(**************************************DIAGNOSTICS**************************************)
(**************************************DIAGNOSTICS**************************************)
(**************************************DIAGNOSTICS**************************************)
	220:// Set Parameters to read the Diagnostic data of the AX5805.		
		IF i_nChooseChannel=1 THEN
			fbCoERead.nSubIndex:=16#07;
		ELSIF
			i_nChooseChannel=2 THEN
			fbCoERead.nSubIndex:=16#08;
		END_IF
		
			fbCoERead.nIndex	:= 	16#FA10;
			fbCoERead.pDstBuf	:= 	ADR(q_stAX5805_Diag.iDiagIndex);
			fbCoERead.cbBufLen	:= 	SIZEOF(q_stAX5805_Diag.iDiagIndex);
			fbCoERead.bExecute	:= 	TRUE;
			iState := iState + 10;	
			
	230:// Evaluate the Diagnostic data of the AX5805.		
		IF NOT fbCoERead.bBusy THEN
			IF q_stAX5805_Diag.iDiagIndex= 0 THEN
				q_stAX5805_Diag.sDiagReaction:='No Error Reaction.';
				ELSIF (q_stAX5805_Diag.iDiagIndex.4 AND q_stAX5805_Diag.iDiagIndex.6) THEN
					q_stAX5805_Diag.sDiagReaction:='SS1 (Safe Stop 1).';
				ELSIF q_stAX5805_Diag.iDiagIndex.6 THEN
					q_stAX5805_Diag.sDiagReaction:='STO (Safe Torque Off).';
				ELSE
					q_stAX5805_Diag.sDiagReaction:='Unknown.';
			END_IF
			
			IF q_stAX5805_Diag.iDiagIndex<255 THEN
				q_stAX5805_Diag.sDiagReason:='No error.';
				ELSIF (q_stAX5805_Diag.iDiagIndex.8 AND q_stAX5805_Diag.iDiagIndex.12 AND q_stAX5805_Diag.iDiagIndex.14 AND q_stAX5805_Diag.iDiagIndex.15) THEN
					q_stAX5805_Diag.sDiagReason:='The Safety Function SDIn has been turned off.';
				ELSIF (q_stAX5805_Diag.iDiagIndex.12 AND q_stAX5805_Diag.iDiagIndex.14 AND q_stAX5805_Diag.iDiagIndex.15) THEN
					q_stAX5805_Diag.sDiagReason:='The Safety Function SDIp has been turned off.';
				ELSIF (q_stAX5805_Diag.iDiagIndex.11 AND q_stAX5805_Diag.iDiagIndex.14 AND q_stAX5805_Diag.iDiagIndex.15) THEN
					q_stAX5805_Diag.sDiagReason:='The Safety Function SMA has been turned off.';
				ELSIF (q_stAX5805_Diag.iDiagIndex.14 AND q_stAX5805_Diag.iDiagIndex.15) THEN
					q_stAX5805_Diag.sDiagReason:='The Safety Function SAR has been turned off.';
				ELSIF (q_stAX5805_Diag.iDiagIndex.11 AND q_stAX5805_Diag.iDiagIndex.12 AND q_stAX5805_Diag.iDiagIndex.13 AND q_stAX5805_Diag.iDiagIndex.15) THEN
					q_stAX5805_Diag.sDiagReason:='The Safety Function SLI has been turned off.';
				ELSIF (q_stAX5805_Diag.iDiagIndex.11 AND q_stAX5805_Diag.iDiagIndex.13 AND q_stAX5805_Diag.iDiagIndex.15) THEN
					q_stAX5805_Diag.sDiagReason:='The Safety Function SMS has been turned off.';
				ELSIF (q_stAX5805_Diag.iDiagIndex.13 AND q_stAX5805_Diag.iDiagIndex.15) THEN
					q_stAX5805_Diag.sDiagReason:='The Safety Function SLP has been turned off.';
				ELSIF (q_stAX5805_Diag.iDiagIndex.12 AND q_stAX5805_Diag.iDiagIndex.15) THEN
					q_stAX5805_Diag.sDiagReason:='The Safety Function SLS has been turned off.';
				ELSIF (q_stAX5805_Diag.iDiagIndex.15) THEN
					q_stAX5805_Diag.sDiagReason:='The Safety Function SSR has been turned off.';
				ELSIF (q_stAX5805_Diag.iDiagIndex.11 AND q_stAX5805_Diag.iDiagIndex.13 AND q_stAX5805_Diag.iDiagIndex.14) THEN
					q_stAX5805_Diag.sDiagReason:='The Safety Function SOS has been turned off.';
				ELSIF (q_stAX5805_Diag.iDiagIndex.12 AND q_stAX5805_Diag.iDiagIndex.14) THEN
					q_stAX5805_Diag.sDiagReason:='The Safety Function SS1 has been turned off.';
				ELSIF (q_stAX5805_Diag.iDiagIndex.11) THEN
					q_stAX5805_Diag.sDiagReason:='The maximum traversing range was exceeded.';
				ELSIF (q_stAX5805_Diag.iDiagIndex.8 AND q_stAX5805_Diag.iDiagIndex.9 AND q_stAX5805_Diag.iDiagIndex.10) THEN
					q_stAX5805_Diag.sDiagReason:='Reason for shutdown position detection: External Cam detected to the left of the cam window.';
				ELSIF (q_stAX5805_Diag.iDiagIndex.9 AND q_stAX5805_Diag.iDiagIndex.10) THEN
					q_stAX5805_Diag.sDiagReason:='Reason for shutdown position detection: External Cam detected to the right of the cam window.';
				ELSIF (q_stAX5805_Diag.iDiagIndex.8 AND q_stAX5805_Diag.iDiagIndex.10) THEN
					q_stAX5805_Diag.sDiagReason:='Reason for shutdown position detection: External Cam detected unexpectedly.';
				ELSIF (q_stAX5805_Diag.iDiagIndex.10) THEN
					q_stAX5805_Diag.sDiagReason:='Internal comparison has failed. Please check the motor and drive dimensioning and parameterization.';
				ELSIF (q_stAX5805_Diag.iDiagIndex.8 AND q_stAX5805_Diag.iDiagIndex.9) THEN
					q_stAX5805_Diag.sDiagReason:='The FSOE Protocol is not in the DATA state.';
				ELSIF (q_stAX5805_Diag.iDiagIndex.9) THEN
					q_stAX5805_Diag.sDiagReason:='The parameters are incorrect or have not been loaded.';
				ELSIF (q_stAX5805_Diag.iDiagIndex.8) THEN
					q_stAX5805_Diag.sDiagReason:='The Status word was calculated incorrectly.';
				ELSIF (i_nChooseChannel<>1 AND i_nChooseChannel<>2) THEN
					q_stAX5805_Diag.sDiagReason:='Wrong Channel Number.';
				ELSE
					q_stAX5805_Diag.sDiagReason:= 'Unknown.';
			END_IF
			
			IF q_stAX5805_Diag.iDiagIndex = 0 THEN
				q_stAX5805_Diag.xDiagnosticAlarm := FALSE;
				ELSE
					q_stAX5805_Diag.xDiagnosticAlarm := TRUE;
			END_IF	
			fbCoERead.bExecute := FALSE;
			q_sErrorDescription := 'No Error';
			iState := iState + 10;
			IF fbCoERead.bError THEN
				q_sErrorDescription := 'AX5805 Diagnostic Data - Read Error';
			END_IF
		END_IF


(**************************************ERRORS**************************************)
(**************************************ERRORS**************************************)
(**************************************ERRORS**************************************)
	240:// Set Parameters to read the Error data of the AX5805.		
		IF i_nChooseChannel=1 THEN
			fbCoERead.nSubIndex:=16#03;
		ELSIF
			i_nChooseChannel=2 THEN
			fbCoERead.nSubIndex:=16#04;
		END_IF
		
			fbCoERead.nIndex	:= 	16#FA82;
			fbCoERead.pDstBuf	:= 	ADR(q_stAX5805_Diag.iErrorIndex);
			fbCoERead.cbBufLen	:= 	SIZEOF(q_stAX5805_Diag.iErrorIndex);
			fbCoERead.bExecute	:= 	TRUE;
			iState := iState + 10;	
			
	250:// Evaluate the Error data of the AX5805.	
		IF NOT fbCoERead.bBusy THEN	
			//0x0000
			IF q_stAX5805_Diag.iErrorIndex = 0 THEN
				q_stAX5805_Diag.sErrorName := 'No Error';
				q_stAX5805_Diag.sErrorDescription := 'No Error';
			//0x0001
			ELSIF q_stAX5805_Diag.iErrorIndex = 16#0001 THEN
				q_stAX5805_Diag.sErrorName := 'FAULT_MAXT_C1';
				q_stAX5805_Diag.sErrorDescription := 'The temperature has exceeded the maximum permissible temperature (MC1).';
				q_stAX5805_Diag.xMC1_TempHighAlarm := TRUE;
			//0x0002
			ELSIF q_stAX5805_Diag.iErrorIndex = 16#0002 THEN
				q_stAX5805_Diag.sErrorName := 'FAULT_MAXT_C2';
				q_stAX5805_Diag.sErrorDescription := 'The temperature has exceeded the maximum permissible temperature (MC2).';
				q_stAX5805_Diag.xMC2_TempHighAlarm := TRUE;
			//0x0003
			ELSIF q_stAX5805_Diag.iErrorIndex = 16#0003 THEN
				q_stAX5805_Diag.sErrorName := 'FAULT_MINT_C1';
				q_stAX5805_Diag.sErrorDescription := 'The temperature has fallen below the minimum permissible temperature (MC1).';
				q_stAX5805_Diag.xMC1_TempLowAlarm := TRUE;
			//0x0004
			ELSIF q_stAX5805_Diag.iErrorIndex = 16#0004 THEN
				q_stAX5805_Diag.sErrorName := 'FAULT_MINT_C2';
				q_stAX5805_Diag.sErrorDescription := 'The temperature has fallen below the minimum permissible temperature (MC2).';
				q_stAX5805_Diag.xMC2_TempLowAlarm := TRUE;	
			//0x0101
			ELSIF q_stAX5805_Diag.iErrorIndex = 16#0101 THEN
				q_stAX5805_Diag.sErrorName := 'HW_ERR_MAX_VCC_C1';
				q_stAX5805_Diag.sErrorDescription := 'The supply voltage has exceeded the maximum permissible voltage MC1 (3.3v).';
				q_stAX5805_Diag.xMC1_SupplyVoltHighAlarm := TRUE;
			//0x0102
			ELSIF q_stAX5805_Diag.iErrorIndex = 16#0102 THEN
				q_stAX5805_Diag.sErrorName := 'HW_ERR_MAX_VCC_C2';
				q_stAX5805_Diag.sErrorDescription := 'The supply voltage has exceeded the maximum permissible voltage MC2 (3.3v).';
				q_stAX5805_Diag.xMC2_SupplyVoltHighAlarm := TRUE;
			//0x0103
			ELSIF q_stAX5805_Diag.iErrorIndex = 16#0103 THEN
				q_stAX5805_Diag.sErrorName := 'HW_ERR_MIN_VCC_C1';
				q_stAX5805_Diag.sErrorDescription := 'The supply voltage has fallen below the minimum permissible voltage MC1 (3.3v).';
				q_stAX5805_Diag.xMC1_SupplyVoltLowAlarm := TRUE;
			//0x0104
			ELSIF q_stAX5805_Diag.iErrorIndex = 16#0104 THEN
				q_stAX5805_Diag.sErrorName := 'HW_ERR_MIN_VCC_C2';
				q_stAX5805_Diag.sErrorDescription := 'The supply voltage has fallen below the minimum permissible voltage MC2 (3.3v).';
				q_stAX5805_Diag.xMC2_SupplyVoltLowAlarm := TRUE;
				
			//0x0201
			ELSIF q_stAX5805_Diag.iErrorIndex = 16#0201 THEN
				q_stAX5805_Diag.sErrorName := 'FAULT_MCTC1_TO';
				q_stAX5805_Diag.sErrorDescription := 'The MCTests of MC1 were not carried out completely within the specified time.';
			//0x0202
			ELSIF q_stAX5805_Diag.iErrorIndex = 16#0202 THEN
				q_stAX5805_Diag.sErrorName := 'FAULT_MCTC2_TO';
				q_stAX5805_Diag.sErrorDescription := 'The MCTests of MC2 were not carried out completely within the specified time.';
			//0x0203
			ELSIF q_stAX5805_Diag.iErrorIndex = 16#0203 THEN
				q_stAX5805_Diag.sErrorName := 'FAULT_TIMER_C1';
				q_stAX5805_Diag.sErrorDescription := 'The global timer was not updated in time MC1.';
			//0x0204
			ELSIF q_stAX5805_Diag.iErrorIndex = 16#0204 THEN
				q_stAX5805_Diag.sErrorName := 'FAULT_TIMER_C2';
				q_stAX5805_Diag.sErrorDescription := 'The global timer was not updated in time MC2.';
			//0x20C
			ELSIF q_stAX5805_Diag.iErrorIndex = 16#020C THEN
				q_stAX5805_Diag.sErrorName := 'FAULT_TS_WDG_TO_C1';
				q_stAX5805_Diag.sErrorDescription := 'The TS module was not called within the watchdog time MC1.';
			//0x020D
			ELSIF q_stAX5805_Diag.iErrorIndex = 16#020D THEN
				q_stAX5805_Diag.sErrorName := 'FAULT_TS_WDG_TO_C2';
				q_stAX5805_Diag.sErrorDescription := 'The TwinSAFE module was not called within the watchdog time MC2.';
			//0x020E
			ELSIF q_stAX5805_Diag.iErrorIndex = 16#020E THEN
				q_stAX5805_Diag.sErrorName := 'FAULT_RESET_MC1';
				q_stAX5805_Diag.sErrorDescription := 'A reset has occurred in the operation of the controller for MC1. MC2 was not reset thereby.';
				
			//0x0300
			ELSIF q_stAX5805_Diag.iErrorIndex = 16#0300 THEN
				q_stAX5805_Diag.sErrorName := 'FAULT_SERCOMC2';
				q_stAX5805_Diag.sErrorDescription := 'Error group: an error occurred in the SerComP24C2 module during data transmission.';
				
			//0x0401
			ELSIF q_stAX5805_Diag.iErrorIndex = 16#0401 THEN
				q_stAX5805_Diag.sErrorName := 'FAULT_SERCOM';
				q_stAX5805_Diag.sErrorDescription := 'Error group: an error occurred in the SerComP24C1 module during data transmission.';
			//0x0402
			ELSIF q_stAX5805_Diag.iErrorIndex = 16#0402 THEN
				q_stAX5805_Diag.sErrorName := 'FAULT_SERCOM';
				q_stAX5805_Diag.sErrorDescription := 'Error group: an error occurred in the SerComP24C1 module during data transmission.';
			//0x0403
			ELSIF q_stAX5805_Diag.iErrorIndex = 16#0403 THEN
				q_stAX5805_Diag.sErrorName := 'FAULT_SERCOM';
				q_stAX5805_Diag.sErrorDescription := 'Error group: an error occurred in the SerComP24C1 module during data transmission.';
			//0x0404
			ELSIF q_stAX5805_Diag.iErrorIndex = 16#0404 THEN
				q_stAX5805_Diag.sErrorName := 'FAULT_SERCOM';
				q_stAX5805_Diag.sErrorDescription := 'Error group: an error occurred in the SerComP24C1 module during data transmission.';
			//0x0405
			ELSIF q_stAX5805_Diag.iErrorIndex = 16#0405 THEN
				q_stAX5805_Diag.sErrorName := 'FAULT_SERCOM';
				q_stAX5805_Diag.sErrorDescription := 'Error group: an error occurred in the SerComP24C1 module during data transmission.';
			//0x0406
			ELSIF q_stAX5805_Diag.iErrorIndex = 16#0406 THEN
				q_stAX5805_Diag.sErrorName := 'FAULT_SERCOM';
				q_stAX5805_Diag.sErrorDescription := 'Error group: an error occurred in the SerComP24C1 module during data transmission.';
			//0x0407
			ELSIF q_stAX5805_Diag.iErrorIndex = 16#0407 THEN
				q_stAX5805_Diag.sErrorName := 'FAULT_SERCOM';
				q_stAX5805_Diag.sErrorDescription := 'Error group: an error occurred in the SerComP24C1 module during data transmission.';
			//0x0408
			ELSIF q_stAX5805_Diag.iErrorIndex = 16#0408 THEN
				q_stAX5805_Diag.sErrorName := 'FAULT_SERCOM';
				q_stAX5805_Diag.sErrorDescription := 'Error group: an error occurred in the SerComP24C1 module during data transmission.';
			//0x0409
			ELSIF q_stAX5805_Diag.iErrorIndex = 16#0409 THEN
				q_stAX5805_Diag.sErrorName := 'FAULT_SERCOM';
				q_stAX5805_Diag.sErrorDescription := 'Error group: an error occurred in the SerComP24C1 module during data transmission.';
			//0x040A
			ELSIF q_stAX5805_Diag.iErrorIndex = 16#040A THEN
				q_stAX5805_Diag.sErrorName := 'FAULT_SERCOM';
				q_stAX5805_Diag.sErrorDescription := 'Error group: an error occurred in the SerComP24C1 module during data transmission.';
			//0x040B
			ELSIF q_stAX5805_Diag.iErrorIndex = 16#040B THEN
				q_stAX5805_Diag.sErrorName := 'FAULT_SERCOM';
				q_stAX5805_Diag.sErrorDescription := 'Error group: an error occurred in the SerComP24C1 module during data transmission.';
			//0x0501
			ELSIF q_stAX5805_Diag.iErrorIndex = 16#0501 THEN
				q_stAX5805_Diag.sErrorName := 'FAULT_TEMPSENSOR';
				q_stAX5805_Diag.sErrorDescription := 'Error in the communication with one of the temperature sensors.';
			//0x0502
			ELSIF q_stAX5805_Diag.iErrorIndex = 16#0502 THEN
				q_stAX5805_Diag.sErrorName := 'FAULT_TEMPSENSOR';
				q_stAX5805_Diag.sErrorDescription := 'Error in the communication with one of the temperature sensors.';
			//0x0503
			ELSIF q_stAX5805_Diag.iErrorIndex = 16#0503 THEN
				q_stAX5805_Diag.sErrorName := 'FAULT_TEMPSENSOR';
				q_stAX5805_Diag.sErrorDescription := 'Error in the communication with one of the temperature sensors..';
			//0x0504
			ELSIF q_stAX5805_Diag.iErrorIndex = 16#0504 THEN
				q_stAX5805_Diag.sErrorName := 'FAULT_TEMPSENSOR';
				q_stAX5805_Diag.sErrorDescription := 'Error in the communication with one of the temperature sensors.';
			//0x0505
			ELSIF q_stAX5805_Diag.iErrorIndex = 16#0505 THEN
				q_stAX5805_Diag.sErrorName := 'FAULT_TEMPSENSOR';
				q_stAX5805_Diag.sErrorDescription := 'Error in the communication with one of the temperature sensors.';
			//0x0506
			ELSIF q_stAX5805_Diag.iErrorIndex = 16#0506 THEN
				q_stAX5805_Diag.sErrorName := 'FAULT_TEMPSENSOR';
				q_stAX5805_Diag.sErrorDescription := 'Error in the communication with one of the temperature sensors.';
			//0x0507
			ELSIF q_stAX5805_Diag.iErrorIndex = 16#0507 THEN
				q_stAX5805_Diag.sErrorName := 'FAULT_TEMPSENSOR';
				q_stAX5805_Diag.sErrorDescription := 'Error in the communication with one of the temperature sensors.';
			//0x0601
			ELSIF q_stAX5805_Diag.iErrorIndex = 16#0601 THEN
				q_stAX5805_Diag.sErrorName := 'FAULT_OUTPUTCOMPARE';
				q_stAX5805_Diag.sErrorDescription := 'The values output by MC1 and MC2 differ.';
			//0x0602
			ELSIF q_stAX5805_Diag.iErrorIndex = 16#0602 THEN
				q_stAX5805_Diag.sErrorName := 'FAULT_OUTPUTCOMPAREC2';
				q_stAX5805_Diag.sErrorDescription := 'The values output by MC1 and MC2 differ.';
			//0x0700
			ELSIF q_stAX5805_Diag.iErrorIndex = 16#0700 THEN
				q_stAX5805_Diag.sErrorName := 'HW_ERR_MIN_VCC_FPGA';
				q_stAX5805_Diag.sErrorDescription := 'The FPGA supply voltage has fallen below the minimum value (5v).';
			//0x0701
			ELSIF q_stAX5805_Diag.iErrorIndex = 16#0701 THEN
				q_stAX5805_Diag.sErrorName := 'HW_ERR_MAX_VCC_FPGA';
				q_stAX5805_Diag.sErrorDescription := 'The FPGA supply voltage has exceeded the maximum value (5v).';
			//0x0710
			ELSIF q_stAX5805_Diag.iErrorIndex = 16#0710 THEN
				q_stAX5805_Diag.sErrorName := 'FAULT_FEEDBACK_C1';
				q_stAX5805_Diag.sErrorDescription := 'An error was detected in the feedback channels of MC1.';
			//0x0711
			ELSIF q_stAX5805_Diag.iErrorIndex = 16#0711 THEN
				q_stAX5805_Diag.sErrorName := 'FAULT_FEEDBACK_C2';
				q_stAX5805_Diag.sErrorDescription := 'An error was detected in the feedback channels of MC2.';
			//0x0720
			ELSIF q_stAX5805_Diag.iErrorIndex = 16#0720 THEN
				q_stAX5805_Diag.sErrorName := 'FAULT_Parameter_C1';
				q_stAX5805_Diag.sErrorDescription := 'General parameter error MC1.';
			//0x0721
			ELSIF q_stAX5805_Diag.iErrorIndex = 16#0721 THEN
				q_stAX5805_Diag.sErrorName := 'FAULT_Parameter_C2';
				q_stAX5805_Diag.sErrorDescription := 'General parameter error MC2.';
			//0x0722
			ELSIF q_stAX5805_Diag.iErrorIndex = 16#0722 THEN
				q_stAX5805_Diag.sErrorName := 'FAULT_Parameter_C1_DRIVE_PROFILE';
				q_stAX5805_Diag.sErrorDescription := 'Parameter: unkown parameter index MC1 drive profile.';
			//0x0723
			ELSIF q_stAX5805_Diag.iErrorIndex = 16#0723 THEN
				q_stAX5805_Diag.sErrorName := 'FAULT_Parameter_C1_VENDOR_SPECIFIC';
				q_stAX5805_Diag.sErrorDescription := 'Parameter: unkown parameter index MC1 vendor-specific.';
			//0x0724
			ELSIF q_stAX5805_Diag.iErrorIndex = 16#0724 THEN
				q_stAX5805_Diag.sErrorName := 'FAULT_Parameter_C2_DRIVE_PROFILE';
				q_stAX5805_Diag.sErrorDescription := 'Parameter: unkown parameter index MC2 drive profile.';
			//0x0725
			ELSIF q_stAX5805_Diag.iErrorIndex = 16#0725 THEN
				q_stAX5805_Diag.sErrorName := 'FAULT_Parameter_C1_VENDOR_SPECIFIC';
				q_stAX5805_Diag.sErrorDescription := 'Parameter: unkown parameter index MC2 vendor-specific.';
			//0x0726
			ELSIF q_stAX5805_Diag.iErrorIndex = 16#0726 THEN
				q_stAX5805_Diag.sErrorName := 'FAULT_DPO_MAPPING_FSOE_COMMAND';
				q_stAX5805_Diag.sErrorDescription := 'PDO mapping: PDO mapping axis 1/2: FSOE COMMAND error.';
			//0x0727
			ELSIF q_stAX5805_Diag.iErrorIndex = 16#0727 THEN
				q_stAX5805_Diag.sErrorName := 'FAULT_PDO_MAPPING_LENGTH';
				q_stAX5805_Diag.sErrorDescription := 'PDO mapping axis 1: Length error.';
			//0x0728
			ELSIF q_stAX5805_Diag.iErrorIndex = 16#0728 THEN
				q_stAX5805_Diag.sErrorName := 'FAULT_PDO_MAPPING_STO_K1';
				q_stAX5805_Diag.sErrorDescription := 'PDO mapping axis 1: STO error.';
			//0x0729
			ELSIF q_stAX5805_Diag.iErrorIndex = 16#0729 THEN
				q_stAX5805_Diag.sErrorName := 'FAULT_PDO_MAPPING_SS1_1_K1';
				q_stAX5805_Diag.sErrorDescription := 'PDO mapping axis 1: Error SS1_1.';
			//0x072A
			ELSIF q_stAX5805_Diag.iErrorIndex = 16#072A THEN
				q_stAX5805_Diag.sErrorName := 'FAULT_PDO_MAPPING_SS2_1_K1';
				q_stAX5805_Diag.sErrorDescription := 'PDO mapping axis 1: Error SS2_1.';
			//0x072B
			ELSIF q_stAX5805_Diag.iErrorIndex = 16#072B THEN
				q_stAX5805_Diag.sErrorName := 'FAULT_PDO_MAPPING_SOS1_K1';
				q_stAX5805_Diag.sErrorDescription := 'PDO mapping axis 1: SOS_1 error.';
			//0x072C
			ELSIF q_stAX5805_Diag.iErrorIndex = 16#072C THEN
				q_stAX5805_Diag.sErrorName := 'FAULT_PDO_MAPPING_SSR_1_K1';
				q_stAX5805_Diag.sErrorDescription := 'PDO mapping axis 1: SSR_1 error.';
			//0x072D
			ELSIF q_stAX5805_Diag.iErrorIndex = 16#072D THEN
				q_stAX5805_Diag.sErrorName := 'FAULT_PDO_MAPPING_SDIp_K1';
				q_stAX5805_Diag.sErrorDescription := 'PDO mapping axis 1: SDIp error.';
			//0x072E
			ELSIF q_stAX5805_Diag.iErrorIndex = 16#072E THEN
				q_stAX5805_Diag.sErrorName := 'FAULT_PDO_MAPPING_SDIn_K1';
				q_stAX5805_Diag.sErrorDescription := 'PDO mapping axis 1: SDIn error.';
			//0x072F
			ELSIF q_stAX5805_Diag.iErrorIndex = 16#072F THEN
				q_stAX5805_Diag.sErrorName := 'FAULT_PDO_MAPPING_Error_ACK_K1';
				q_stAX5805_Diag.sErrorDescription := 'PDO mapping axis 1: Error_ACK error.';
			//0X0730
			ELSIF q_stAX5805_Diag.iErrorIndex = 16#0730 THEN
				q_stAX5805_Diag.sErrorName := 'FAULT_PDO_MAPPING_Error_CRC0';
				q_stAX5805_Diag.sErrorDescription := 'PDO mapping axis 1/2: FSOE CRC0 error.';
			//0x0731
			ELSIF q_stAX5805_Diag.iErrorIndex = 16#0731 THEN
				q_stAX5805_Diag.sErrorName := 'FAULT_PDO_MAPPING_STO_K2';
				q_stAX5805_Diag.sErrorDescription := 'PDO mapping axis 2: STO error.';
			//0x0732
			ELSIF q_stAX5805_Diag.iErrorIndex = 16#0732 THEN
				q_stAX5805_Diag.sErrorName := 'FAULT_PDO_MAPPING_SS1_2_K2';
				q_stAX5805_Diag.sErrorDescription := 'PDO mapping axis 2: Error SS1_1.';
			//0x0733
			ELSIF q_stAX5805_Diag.iErrorIndex = 16#0733 THEN
				q_stAX5805_Diag.sErrorName := 'FAULT_PDO_MAPPING_SS2_1_K2';
				q_stAX5805_Diag.sErrorDescription := 'PDO mapping axis 2: Error SS2_1.';
			//0x0734
			ELSIF q_stAX5805_Diag.iErrorIndex = 16#0734 THEN
				q_stAX5805_Diag.sErrorName := 'FAULT_PDO_MAPPING_SOS_1_K2';
				q_stAX5805_Diag.sErrorDescription := 'PDO mapping axis 2: SOS_1 error.';
			//0x0735
			ELSIF q_stAX5805_Diag.iErrorIndex = 16#0735 THEN
				q_stAX5805_Diag.sErrorName := 'FAULT_PDO_MAPPING_SSR_1_K2';
				q_stAX5805_Diag.sErrorDescription := 'PDO mapping axis 2: SSR_1 error.';
			//0x0736
			ELSIF q_stAX5805_Diag.iErrorIndex = 16#0736 THEN
				q_stAX5805_Diag.sErrorName := 'FAULT_PDO_MAPPING_SDIp_K2';
				q_stAX5805_Diag.sErrorDescription := 'PDO mapping axis 2: SDIp error.';
			//0x0737
			ELSIF q_stAX5805_Diag.iErrorIndex = 16#0737 THEN
				q_stAX5805_Diag.sErrorName := 'FAULT_PDO_MAPPING_SDIn_K2';
				q_stAX5805_Diag.sErrorDescription := 'PDO mapping axis 2: SDIn error.';
			//0x0738
			ELSIF q_stAX5805_Diag.iErrorIndex = 16#0738 THEN
				q_stAX5805_Diag.sErrorName := 'FAULT_PDO_MAPPING_Error_ACK_K2';
				q_stAX5805_Diag.sErrorDescription := 'PDO mapping axis 2: Error_ACK error.';
			//0x0739
			ELSIF q_stAX5805_Diag.iErrorIndex = 16#0739 THEN
				q_stAX5805_Diag.sErrorName := 'FAULT_PDO_MAPPING_Error_CRC1';
				q_stAX5805_Diag.sErrorDescription := 'PDO mapping axis 2: FSOE CRC1 error.';
			//0x073A
			ELSIF q_stAX5805_Diag.iErrorIndex = 16#073A THEN
				q_stAX5805_Diag.sErrorName := 'FAULT_PDO_MAPPING_Error_ConnID';
				q_stAX5805_Diag.sErrorDescription := 'PDO mapping axis 1/2: FSOE ConnID error.';
			//0x073B
			ELSIF q_stAX5805_Diag.iErrorIndex = 16#073B THEN
				q_stAX5805_Diag.sErrorName := 'FAULT_PDO_MAPPING_SSM_1_K1';
				q_stAX5805_Diag.sErrorDescription := 'PDO mapping axis 1: SSM_1_K1 error.';
			//0x073C
			ELSIF q_stAX5805_Diag.iErrorIndex = 16#073C THEN
				q_stAX5805_Diag.sErrorName := 'FAULT_PDO_MAPPING_SSM_1_K2';
				q_stAX5805_Diag.sErrorDescription := 'PDO mapping axis 2: SSM_1_K2 error.';
			//0x073D
			ELSIF q_stAX5805_Diag.iErrorIndex = 16#073D THEN
				q_stAX5805_Diag.sErrorName := 'FAULT_PDO_MAPPING_SSM2_K1';
				q_stAX5805_Diag.sErrorDescription := 'PDO mapping axis 1: SSM_2_K1 error.';
			//0x073E
			ELSIF q_stAX5805_Diag.iErrorIndex = 16#073E THEN
				q_stAX5805_Diag.sErrorName := 'FAULT_PDO_MAPPING_SSM2_K2';
				q_stAX5805_Diag.sErrorDescription := 'PDO mapping axis 2: SSM_2_K2 error.';
			//0X740
			ELSIF q_stAX5805_Diag.iErrorIndex = 16#0740 THEN
				q_stAX5805_Diag.sErrorName := 'FAULT_WRONG_MOTORCONTRUCTIONTYPE_K1';
				q_stAX5805_Diag.sErrorDescription := 'Register communication: Parameterized motor type for Axis 1 does not corresopond to the connected motor.';
			//0x0741
			ELSIF q_stAX5805_Diag.iErrorIndex = 16#0741 THEN
				q_stAX5805_Diag.sErrorName := 'FAULT_UNKNOWN_MOTOR_TYPE_K1';
				q_stAX5805_Diag.sErrorDescription := 'Register communication: Parameterized motor type for Axis 1 is unknown.';
			//0x0742
			ELSIF q_stAX5805_Diag.iErrorIndex = 16#0742 THEN
				q_stAX5805_Diag.sErrorName := 'FAULT_WRONG_MOTORCONSTRUCTIONTYPE_K2';
				q_stAX5805_Diag.sErrorDescription := 'Register communication: Parameterized motor type for Axis 2 does not corresopond to the connected motor.';
			//0x0743
			ELSIF q_stAX5805_Diag.iErrorIndex = 16#0743 THEN
				q_stAX5805_Diag.sErrorName := 'FAULT_UNKNOWN_MOTOR_TYPE_K2';
				q_stAX5805_Diag.sErrorDescription := 'Register communication: Parameterized motor type for Axis 2 is unknown.';
			//0x0744
			ELSIF q_stAX5805_Diag.iErrorIndex = 16#0744 THEN
				q_stAX5805_Diag.sErrorName := 'FAULT_NUM_OF_POLEPAIRS_K1';
				q_stAX5805_Diag.sErrorDescription := 'Register communication: Parameterized number of pole pairs for Axis 1 does not corresopond to the connected motor.';
			//0x0745
			ELSIF q_stAX5805_Diag.iErrorIndex = 16#0745 THEN
				q_stAX5805_Diag.sErrorName := 'FAULT_NUM_OF_POLEPAIRS_K2';
				q_stAX5805_Diag.sErrorDescription := 'Register communication: Parameterized number of pole pairs for Axis 2 does not corresopond to the connected motor.';
			//0x0746
			ELSIF q_stAX5805_Diag.iErrorIndex = 16#0746 THEN
				q_stAX5805_Diag.sErrorName := 'FAULT_WRONG_MOTOR_CONFIGURED_K1';
				q_stAX5805_Diag.sErrorDescription := 'Register communication: Parameterized motor type for Axis 1 does not corresopond to the connected motor.';
			//0x0747
			ELSIF q_stAX5805_Diag.iErrorIndex = 16#0747 THEN
				q_stAX5805_Diag.sErrorName := 'FAULT_WRONG_MOTOR_CONFIGURED_K2';
				q_stAX5805_Diag.sErrorDescription := 'Register communication: Parameterized motor type for Axis 2 does not corresopond to the connected motor.';	
			//0x0748
			ELSIF q_stAX5805_Diag.iErrorIndex = 16#0748 THEN
				q_stAX5805_Diag.sErrorName := 'FAULT_RXPDO_LENGTH';
				q_stAX5805_Diag.sErrorDescription := 'PDO mapping: RXPDO length is wrong.';
			//0x0749
			ELSIF q_stAX5805_Diag.iErrorIndex = 16#0749 THEN
				q_stAX5805_Diag.sErrorName := 'FAULT_TXPDO_LENGTH';
				q_stAX5805_Diag.sErrorDescription := 'PDO mapping: TXPDO length is wrong.';
			//0x074A
			ELSIF q_stAX5805_Diag.iErrorIndex = 16#074A THEN
				q_stAX5805_Diag.sErrorName := 'FAULT_UNKNOWN_RXPDO_INDEX';
				q_stAX5805_Diag.sErrorDescription := 'PDO mapping: RXPDO index is unknown.';
			//0x074B
			ELSIF q_stAX5805_Diag.iErrorIndex = 16#074B THEN
				q_stAX5805_Diag.sErrorName := 'FAULT_UNKNOWN_TXPDO_INDEX';
				q_stAX5805_Diag.sErrorDescription := 'PDO mapping: TXPDO index is unknown.';
			//0x074C
			ELSIF q_stAX5805_Diag.iErrorIndex = 16#074C THEN
				q_stAX5805_Diag.sErrorName := 'FAULT_WRONG_NUMBER_OF_AXLE';
				q_stAX5805_Diag.sErrorDescription := 'The parameterized number of axes does not correspond to the number detected.';
			//1001
			ELSIF q_stAX5805_Diag.iErrorIndex = 16#1001 THEN
				q_stAX5805_Diag.sErrorName := 'FAULT_CRC_INIT_C1';
				q_stAX5805_Diag.sErrorDescription := 'An incorrect checksum was determined for MC1 during PowerOn reset.';
			//0x1002
			ELSIF q_stAX5805_Diag.iErrorIndex = 16#1002 THEN
				q_stAX5805_Diag.sErrorName := 'FAULT_CRC_INIT_C2';
				q_stAX5805_Diag.sErrorDescription := 'An incorrect checksum was determined for MC2 during PowerOn reset.';
			//0x1003
			ELSIF q_stAX5805_Diag.iErrorIndex = 16#1003 THEN
				q_stAX5805_Diag.sErrorName := 'FAULT_CRC_C1';
				q_stAX5805_Diag.sErrorDescription := 'An incorrect checksum was determined for MC1 during operation.';
			//0x1004
			ELSIF q_stAX5805_Diag.iErrorIndex = 16#1004 THEN
				q_stAX5805_Diag.sErrorName := 'FAULT_CRC_C2';
				q_stAX5805_Diag.sErrorDescription := 'An incorrect checksum was determined for MC2 during operation.';
			//0X1011
			ELSIF q_stAX5805_Diag.iErrorIndex = 16#1011 THEN
				q_stAX5805_Diag.sErrorName := 'FAULT_RAM_C1';
				q_stAX5805_Diag.sErrorDescription := 'An error occurred during the RAM test of MC1.';
			//0x1012
			ELSIF q_stAX5805_Diag.iErrorIndex = 16#1012 THEN
				q_stAX5805_Diag.sErrorName := 'FAULT_RAM_C2';
				q_stAX5805_Diag.sErrorDescription := 'An error occurred during the RAM test of MC2.';
			//0x1013
			ELSIF q_stAX5805_Diag.iErrorIndex = 16#1013 THEN
				q_stAX5805_Diag.sErrorName := 'FAULT_RAM_CHECKERBOARD_C1';
				q_stAX5805_Diag.sErrorDescription := 'An error occurred during the RAM test of MC1.';
			//0x1014
			ELSIF q_stAX5805_Diag.iErrorIndex = 16#1014 THEN
				q_stAX5805_Diag.sErrorName := 'FAULT_RAM_CHECKERBOARD_C2';
				q_stAX5805_Diag.sErrorDescription := 'An error occurred during the RAM test of MC2.';
			//0X1021
			ELSIF q_stAX5805_Diag.iErrorIndex = 16#1021 THEN
				q_stAX5805_Diag.sErrorName := 'FAULT_GLBL_TMR';
				q_stAX5805_Diag.sErrorDescription := 'The global timer is not working correctly.';
			//0X1031
			ELSIF q_stAX5805_Diag.iErrorIndex = 16#1022 THEN
				q_stAX5805_Diag.sErrorName := 'FAULT_SPLIM1';
				q_stAX5805_Diag.sErrorDescription := 'Stack overruns are no longer being intercepted correctly.';
			//0x1032
			ELSIF q_stAX5805_Diag.iErrorIndex = 16#1032 THEN
				q_stAX5805_Diag.sErrorName := 'FAULT_SPLIM2';
				q_stAX5805_Diag.sErrorDescription := 'Stack overruns are no longer being intercepted correctly.';
			//1100
			ELSIF q_stAX5805_Diag.iErrorIndex = 16#1100 THEN
				q_stAX5805_Diag.sErrorName := 'FAULT_OPCT_GRP_C1';
				q_stAX5805_Diag.sErrorDescription := 'The Opcode test for MC1 has failed.';
			//0X1300
			ELSIF q_stAX5805_Diag.iErrorIndex = 16#1300 THEN
				q_stAX5805_Diag.sErrorName := 'FAULT_OPCT_GRP_C2';
				q_stAX5805_Diag.sErrorDescription := 'The Opcode test for MC2 has failed.';
			//0X1801
			ELSIF q_stAX5805_Diag.iErrorIndex = 16#1801 THEN
				q_stAX5805_Diag.sErrorName := 'FAULT_ESS_CRC_C1';
				q_stAX5805_Diag.sErrorDescription := 'Different check sums were determined in the TwinSAFE telegrames MC1.';
			//0x1802
			ELSIF q_stAX5805_Diag.iErrorIndex = 16#1802 THEN
				q_stAX5805_Diag.sErrorName := 'FAULT_ESS_CRC_C2';
				q_stAX5805_Diag.sErrorDescription := 'Different check sums were determined in the TwinSAFE telegrames MC2.';
			//0x1803
			ELSIF q_stAX5805_Diag.iErrorIndex = 16#1803 THEN
				q_stAX5805_Diag.sErrorName := 'FAULT_SW_MAIN1_C1';
				q_stAX5805_Diag.sErrorDescription := 'The default case of the main loop of MC1 was called.';
			//0x1804
			ELSIF q_stAX5805_Diag.iErrorIndex = 16#1804 THEN
				q_stAX5805_Diag.sErrorName := 'FAULT_SW_MAIN1_C2';
				q_stAX5805_Diag.sErrorDescription := 'The default case of the main loop of MC2 was called.';
			//0x1805
			ELSIF q_stAX5805_Diag.iErrorIndex = 16#1805 THEN
				q_stAX5805_Diag.sErrorName := 'FAULT_ESLCONID_PRJCRCRD';
				q_stAX5805_Diag.sErrorDescription := 'The Connection ID is not zero when reading the project CRC.';
			//0x1806
			ELSIF q_stAX5805_Diag.iErrorIndex = 16#1806 THEN
				q_stAX5805_Diag.sErrorName := 'FAULT_ESLCONID_PRJCRCWR';
				q_stAX5805_Diag.sErrorDescription := 'The Connection ID is not zero when writing the project CRC.';
			//0x1807
			ELSIF q_stAX5805_Diag.iErrorIndex = 16#1807 THEN
				q_stAX5805_Diag.sErrorName := 'FAULT_SIZE_EEVONDOR_EXID';
				q_stAX5805_Diag.sErrorDescription := 'An address was accessed theat lies outside the vendor range in the EEPROM.';
			//0X5100
			ELSIF q_stAX5805_Diag.iErrorIndex = 16#5100 THEN
				q_stAX5805_Diag.sErrorName := 'FAULT_COM_C1C2';
				q_stAX5805_Diag.sErrorDescription := 'Communication between MC1 and MC2 is disturbed.';	
			//0X5101
			ELSIF q_stAX5805_Diag.iErrorIndex = 16#5101 THEN
				q_stAX5805_Diag.sErrorName := 'FAULT_ISR_SNT_FEEDBACK';
				q_stAX5805_Diag.sErrorDescription := 'High priority ISR: communication interrupted: switched mode power supply feedback.';	
			//0X5102
			ELSIF q_stAX5805_Diag.iErrorIndex = 16#5102 THEN
				q_stAX5805_Diag.sErrorName := 'FAULT_ISR_ANGLE_K1';
				q_stAX5805_Diag.sErrorDescription := 'High priority ISR: communication interrupted: axis 1 angle.';	
			//0X5103
			ELSIF q_stAX5805_Diag.iErrorIndex = 16#5103 THEN
				q_stAX5805_Diag.sErrorName := 'FAULT_IRS_ANGLE_K2';
				q_stAX5805_Diag.sErrorDescription := 'High priority ISR: communication interrupted: axis 2 angle.';	
			//0X5104
			ELSIF q_stAX5805_Diag.iErrorIndex = 16#5104 THEN
				q_stAX5805_Diag.sErrorName := 'FAULT_ISR_DELTA_K1';
				q_stAX5805_Diag.sErrorDescription := 'High priority ISR: communication interrupted: axis 1 distance travelled.';	
			//0X5105
			ELSIF q_stAX5805_Diag.iErrorIndex = 16#5105 THEN
				q_stAX5805_Diag.sErrorName := 'FAULT_ISR_DELTA_K2';
				q_stAX5805_Diag.sErrorDescription := 'High priority ISR: communication interrupted: axis 2 distance travelled.';	
			//0X5106
			ELSIF q_stAX5805_Diag.iErrorIndex = 16#5106 THEN
				q_stAX5805_Diag.sErrorName := 'FAULT_ISR_VELO_K1';
				q_stAX5805_Diag.sErrorDescription := 'High priority ISR: communication interrupted: axis 1 velocity.';	
			//0X5107
			ELSIF q_stAX5805_Diag.iErrorIndex = 16#5107 THEN
				q_stAX5805_Diag.sErrorName := 'FAULT_ISR_VELO_K2';
				q_stAX5805_Diag.sErrorDescription := 'High priority ISR: communication interrupted: axis 2 velocity.';	
			//0X5108
			ELSIF q_stAX5805_Diag.iErrorIndex = 16#5108 THEN
				q_stAX5805_Diag.sErrorName := 'FAULT_ISR_TEST_FEEDBACK';
				q_stAX5805_Diag.sErrorDescription := 'High priority ISR: communication interrupted: feedback from switch-off channels.';	
			//0X5109
			ELSIF q_stAX5805_Diag.iErrorIndex = 16#5109 THEN
				q_stAX5805_Diag.sErrorName := 'FAULT_TIMEOUT_REG_AX5000_CONTROL';
				q_stAX5805_Diag.sErrorDescription := 'High priority ISR: AX5000 des not answer in time: Control word.';	
			//0X510A
			ELSIF q_stAX5805_Diag.iErrorIndex = 16#510A THEN
				q_stAX5805_Diag.sErrorName := 'FAULT_TIMEOUT_REG_AX5000_STATUS';
				q_stAX5805_Diag.sErrorDescription := 'High priority ISR: AX5000 des not answer in time: Status word.';	
			//0X510B
			ELSIF q_stAX5805_Diag.iErrorIndex = 16#510B THEN
				q_stAX5805_Diag.sErrorName := 'FAULT_TIMEOUT_REG_AX5000_REGADR';
				q_stAX5805_Diag.sErrorDescription := 'High priority ISR: AX5000 des not answer in time: Register address.';	
			//0X510C
			ELSIF q_stAX5805_Diag.iErrorIndex = 16#510C THEN
				q_stAX5805_Diag.sErrorName := 'FAULT_TIMEOUT_REG_AX5000_REGDATA';
				q_stAX5805_Diag.sErrorDescription := 'High priority ISR: AX5000 des not answer in time: Register data.';	
			//0X510D
			ELSIF q_stAX5805_Diag.iErrorIndex = 16#510D THEN
				q_stAX5805_Diag.sErrorName := 'FAULT_TIMEOUT_REG_AX5000_CRC';
				q_stAX5805_Diag.sErrorDescription := 'High priority ISR: AX5000 des not answer in time: CRC.';	
			//0X510E
			ELSIF q_stAX5805_Diag.iErrorIndex = 16#510E THEN
				q_stAX5805_Diag.sErrorName := 'FAULT_UNKNOWN_AX5000_INTERFACE';
				q_stAX5805_Diag.sErrorDescription := 'High priority ISR: Unkown interface to the AX5000.';	
			//0X510F
			ELSIF q_stAX5805_Diag.iErrorIndex = 16#510F THEN
				q_stAX5805_Diag.sErrorName := 'FAULT_COMERROR_AX5000_INTERFACE';
				q_stAX5805_Diag.sErrorDescription := 'High priority ISR: The interface to the AX5000 has a communication error.';
			//0X5110
			ELSIF q_stAX5805_Diag.iErrorIndex = 16#5110 THEN
				q_stAX5805_Diag.sErrorName := 'FAULT_WRITE_HW_VERSION_AX5805';
				q_stAX5805_Diag.sErrorDescription := 'Register communication: Hardware version could not be written to the register in the AX5000.';	
			//0X5111
			ELSIF q_stAX5805_Diag.iErrorIndex = 16#5111 THEN
				q_stAX5805_Diag.sErrorName := 'FAULT_WRITE_HW_VERSION_AX5805';
				q_stAX5805_Diag.sErrorDescription := 'Register communication: Hardware version could not be written to the register in the AX5000.';	
			//0X5112
			ELSIF q_stAX5805_Diag.iErrorIndex = 16#5112 THEN
				q_stAX5805_Diag.sErrorName := 'FAULT_WRITE_HW_VERSION_AX5805';
				q_stAX5805_Diag.sErrorDescription := 'Register communication: Hardware version could not be written to the register in the AX5000.';	
			//0X5113
			ELSIF q_stAX5805_Diag.iErrorIndex = 16#5113 THEN
				q_stAX5805_Diag.sErrorName := 'FAULT_WRITE_HW_VERSION_AX5805';
				q_stAX5805_Diag.sErrorDescription := 'Register communication: Hardware version could not be written to the register in the AX5000.';
			//0X5114
			ELSIF q_stAX5805_Diag.iErrorIndex = 16#5114  THEN
				q_stAX5805_Diag.sErrorName := 'FAULT_EXT_ADC_ADDRESS';
				q_stAX5805_Diag.sErrorDescription := 'High priority ISR: External ADC: An impermissible address was read.';	
			//0X5115
			ELSIF q_stAX5805_Diag.iErrorIndex = 16#5115 THEN
				q_stAX5805_Diag.sErrorName := 'FAULT_REGISTER_AX5000_CRC_ERROR';
				q_stAX5805_Diag.sErrorDescription := 'Register communication with the AX5000: telegram has a CRC error.';	
			//0X5116
			ELSIF q_stAX5805_Diag.iErrorIndex = 16#5116 THEN
				q_stAX5805_Diag.sErrorName := 'FAULT_CYCLIC_AX5000_CRC_ERROR';
				q_stAX5805_Diag.sErrorDescription := 'High priority ISR: Cyclic communication with the AX5000: Telegram has a CRC error.';	
			//0X5117
			ELSIF q_stAX5805_Diag.iErrorIndex = 16#5117 THEN
				q_stAX5805_Diag.sErrorName := 'FAULT_UNKNOWN_REGISTER_ADDRESS';
				q_stAX5805_Diag.sErrorDescription := 'Register communication: Addressed register is unkown.';	
			//0X5118
			ELSIF q_stAX5805_Diag.iErrorIndex = 16#5118 THEN
				q_stAX5805_Diag.sErrorName := 'FAULT_AX5000_NOT_READY';
				q_stAX5805_Diag.sErrorDescription := 'High priority ISR: Cyclic communication with the AX5000: AX5000 signals a communication error.';	
			//0X5119
			ELSIF q_stAX5805_Diag.iErrorIndex = 16#5119 THEN
				q_stAX5805_Diag.sErrorName := 'FAULT_C1C2_SYNC_LOST';
				q_stAX5805_Diag.sErrorDescription := 'High priority ISR: Cyclic communication between MC1 and MC2: Communication error.';
			//0X5C00
			ELSIF q_stAX5805_Diag.iErrorIndex = 16#5C00 THEN
				q_stAX5805_Diag.sErrorName := 'FAULT_SET_MAPPED_STATE';
				q_stAX5805_Diag.sErrorDescription := 'Mapped safety functions: Error while setting the state.';	
			//0X5C01
			ELSIF q_stAX5805_Diag.iErrorIndex = 16#5C01 THEN
				q_stAX5805_Diag.sErrorName := 'FAULT_RESET_MAPPED_STATE';
				q_stAX5805_Diag.sErrorDescription := 'Mapped safety functions: Error while resetting the state.';	
			//0X5C02
			ELSIF q_stAX5805_Diag.iErrorIndex = 16#5C02 THEN
				q_stAX5805_Diag.sErrorName := 'FAULT_MAPPED_FUNCTION';
				q_stAX5805_Diag.sErrorDescription := 'Mapped safety functions: Invalid mapping, function does not exist.';	
			//0X5C03
			ELSIF q_stAX5805_Diag.iErrorIndex = 16#5C03 THEN
				q_stAX5805_Diag.sErrorName := 'FAULT_MAPPED_INSTANCE';
				q_stAX5805_Diag.sErrorDescription := 'Mapped safety functions: Invalid mapping, instance does not exist.';
			//0X5E02
			ELSIF q_stAX5805_Diag.iErrorIndex = 16#5E02 THEN
				q_stAX5805_Diag.sErrorName := 'FAULT_STO_MODE';
				q_stAX5805_Diag.sErrorDescription := 'The requested STO mode is invalid.';	
			//0X5E03
			ELSIF q_stAX5805_Diag.iErrorIndex = 16#5E03 THEN
				q_stAX5805_Diag.sErrorName := 'FAULT_SDI_MODE';
				q_stAX5805_Diag.sErrorDescription := 'The requested SDI mode is invalid.';	
			//0X5E04
			ELSIF q_stAX5805_Diag.iErrorIndex = 16#5E04 THEN
				q_stAX5805_Diag.sErrorName := 'FAULT_UNDEFINED_ERRORREACTION';
				q_stAX5805_Diag.sErrorDescription := 'Error reaction: Invalid error reaction, error reaction does not exist.';	
			//0X5F00
			ELSIF q_stAX5805_Diag.iErrorIndex = 16#5F00 THEN
				q_stAX5805_Diag.sErrorName := 'FAULT_CRC_COMPARE_C1';
				q_stAX5805_Diag.sErrorDescription := 'An incorrect checksum was determined when comparing with MC1.';		
			//0X5F01
			ELSIF q_stAX5805_Diag.iErrorIndex = 16#5F01 THEN
				q_stAX5805_Diag.sErrorName := 'FAULT_CRC_COMPARE_C2';
				q_stAX5805_Diag.sErrorDescription := 'An incorrect checksum was determined when comparing with MC2.';	
			//0X5F02
			ELSIF q_stAX5805_Diag.iErrorIndex = 16#5F02 THEN
				q_stAX5805_Diag.sErrorName := 'FAULT_TMR2_INTERRUPT_C1';
				q_stAX5805_Diag.sErrorDescription := 'MC_Test: Timer2 has triggered an interrupt on MC1. HighPrioISR was not called in time.';	
			//0X5F03
			ELSIF q_stAX5805_Diag.iErrorIndex = 16#5F03 THEN
				q_stAX5805_Diag.sErrorName := 'FAULT_TMR2_INTERRUPT_C2';
				q_stAX5805_Diag.sErrorDescription := 'MC_Test: Timer2 has triggered an interrupt on MC2. HighPrioISR was not called in time.';	
			//0X5F04
			ELSIF q_stAX5805_Diag.iErrorIndex = 16#5F04 THEN
				q_stAX5805_Diag.sErrorName := 'FAULT_SWITCHOFF_TEST';
				q_stAX5805_Diag.sErrorDescription := 'MC_Test: The test of the switch-off channels has failed.';	
			//0X5F05
			ELSIF q_stAX5805_Diag.iErrorIndex = 16#5F05 THEN
				q_stAX5805_Diag.sErrorName := 'FAULT_NO_SYNC';
				q_stAX5805_Diag.sErrorDescription := 'No SYNC signal.';		
			//0X5F06
			ELSIF q_stAX5805_Diag.iErrorIndex = 16#5F06 THEN
				q_stAX5805_Diag.sErrorName := 'FAULT_UNKNOWN_AXLE';
				q_stAX5805_Diag.sErrorDescription := 'The requested axis is unknown.';	
			//0X5F07
			ELSIF q_stAX5805_Diag.iErrorIndex = 16#5F07 THEN
				q_stAX5805_Diag.sErrorName := 'FAULT_FPGA_C2';
				q_stAX5805_Diag.sErrorDescription := 'The status of the FPGA is incorrect.';	
			//0X5F08
			ELSIF q_stAX5805_Diag.iErrorIndex = 16#5F08 THEN
				q_stAX5805_Diag.sErrorName := 'FAULT_ANGLE_FORMAT_C1';
				q_stAX5805_Diag.sErrorDescription := 'The angles of MC1 read-in have the wrong format.';	
			//0X5F09
			ELSIF q_stAX5805_Diag.iErrorIndex = 16#5F09 THEN
				q_stAX5805_Diag.sErrorName := 'FAULT_ANGLE_FORMAT_C2';
				q_stAX5805_Diag.sErrorDescription := 'The angles of MC2 read-in have the wrong format.';	
			//0X5F0A
			ELSIF q_stAX5805_Diag.iErrorIndex = 16#5F0A THEN
				q_stAX5805_Diag.sErrorName := 'FAULT_SAFE_MAIN_STATE';
				q_stAX5805_Diag.sErrorDescription := 'Unkown state requested.';	
			//0X5F0B
			ELSIF q_stAX5805_Diag.iErrorIndex = 16#5F0B THEN
				q_stAX5805_Diag.sErrorName := 'FAULT_STARTUP_FAILED';
				q_stAX5805_Diag.sErrorDescription := 'Error during start-up.';	
			//0X5F0C
			ELSIF q_stAX5805_Diag.iErrorIndex = 16#5F0C THEN
				q_stAX5805_Diag.sErrorName := 'FAULT_MOTION_DETECTION';
				q_stAX5805_Diag.sErrorDescription := 'Motion detection error.';	
			//0X6000
			ELSIF q_stAX5805_Diag.iErrorIndex = 16#6000 THEN
				q_stAX5805_Diag.sErrorName := 'FAULT_PARAMETER_FSOE_VENDOR_ID';
				q_stAX5805_Diag.sErrorDescription := 'Incorrect vendor ID transmitted.';	
			//0X6001
			ELSIF q_stAX5805_Diag.iErrorIndex = 16#6001 THEN
				q_stAX5805_Diag.sErrorName := 'FAULT_PARAMETER_FSOE_MODULE_IDENT';
				q_stAX5805_Diag.sErrorDescription := 'Incorrect module ID transmitted.';	
			//0X6002
			ELSIF q_stAX5805_Diag.iErrorIndex = 16#6002 THEN
				q_stAX5805_Diag.sErrorName := 'FAULT_PARAMETER_FSOE_CRC';
				q_stAX5805_Diag.sErrorDescription := 'CRC of the AX5805 parameters does not match the transmitted CRC.';
			ELSE
				q_stAX5805_Diag.sErrorName := 'ERROR';
				q_stAX5805_Diag.sErrorDescription := 'Unknown Index.';
			END_IF
		
			IF q_stAX5805_Diag.iErrorIndex = 0 THEN
				q_stAX5805_Diag.xErrorAlarm := FALSE;
			ELSE
				q_stAX5805_Diag.xErrorAlarm := TRUE;
			END_IF
			fbCoERead.bExecute := FALSE;
			q_sErrorDescription := 'No Error';
			iState := iState + 10;
			IF fbCoERead.bError THEN
				q_sErrorDescription := 'AX5805 Error Data - Read Error';
			END_IF
		END_IF

	260:// Set Parameters to read the Connection State of the AX5805.		
			fbCoERead.nSubIndex	:= 	1;
			fbCoERead.nIndex	:= 	16#EA00;
			fbCoERead.pDstBuf	:= 	ADR(iAX5805_ConnectionState);
			fbCoERead.cbBufLen	:= 	SIZEOF(iAX5805_ConnectionState);
			fbCoERead.bExecute	:= 	TRUE;
			iState := iState + 10;	
			
	270:// Evaluate the Connection State of the AX5805.		
		IF NOT fbCoERead.bBusy THEN
			IF iAX5805_ConnectionState = 0 THEN
				q_stAX5805_Diag.sConnectionState := 'Reset State';
				ELSIF iAX5805_ConnectionState = 1 THEN
					q_stAX5805_Diag.sConnectionState := 'Session State';
				ELSIF iAX5805_ConnectionState = 2 THEN
					q_stAX5805_Diag.sConnectionState := 'Connection State';
				ELSIF iAX5805_ConnectionState = 3 THEN
					q_stAX5805_Diag.sConnectionState := 'Parameter State';
				ELSIF iAX5805_ConnectionState = 4 THEN
					q_stAX5805_Diag.sConnectionState := 'Data State';
				ELSIF iAX5805_ConnectionState = 5 THEN
					q_stAX5805_Diag.sConnectionState := 'Failsafe State';
				ELSE
					q_stAX5805_Diag.sConnectionState := 'Undefined State';
			END_IF
			fbCoERead.bExecute := FALSE;
			q_sErrorDescription := 'No Error';
			iState := 0;
			IF fbCoERead.bError THEN
				q_sErrorDescription := 'AX5805 Connection State - Read Error';
			END_IF
		END_IF
END_CASE

// If any of above errors exist set q_stAX5805_Diag.xAX5805Error TRUE.
		IF NOT q_stAX5805_Diag.xDiagnosticAlarm OR
			q_stAX5805_Diag.xErrorAlarm OR
			q_stAX5805_Diag.xMC1_SupplyVoltHighAlarm OR
			q_stAX5805_Diag.xMC1_SupplyVoltLowAlarm OR
			q_stAX5805_Diag.xMC1_TempHighAlarm OR
			q_stAX5805_Diag.xMC1_TempLowAlarm OR
			q_stAX5805_Diag.xMC2_SupplyVoltHighAlarm OR
			q_stAX5805_Diag.xMC2_SupplyVoltLowAlarm OR
			q_stAX5805_Diag.xMC2_TempHighAlarm OR
			q_stAX5805_Diag.xMC2_TempLowAlarm THEN
				q_stAX5805_Diag.xAX5805Error := FALSE;
		ELSIF q_stAX5805_Diag.xDiagnosticAlarm OR
			q_stAX5805_Diag.xErrorAlarm OR
			q_stAX5805_Diag.xMC1_SupplyVoltHighAlarm OR
			q_stAX5805_Diag.xMC1_SupplyVoltLowAlarm OR
			q_stAX5805_Diag.xMC1_TempHighAlarm OR
			q_stAX5805_Diag.xMC1_TempLowAlarm OR
			q_stAX5805_Diag.xMC2_SupplyVoltHighAlarm OR
			q_stAX5805_Diag.xMC2_SupplyVoltLowAlarm OR
			q_stAX5805_Diag.xMC2_TempHighAlarm OR
			q_stAX5805_Diag.xMC2_TempLowAlarm THEN
				q_stAX5805_Diag.xAX5805Error := TRUE;
		END_IF

// FB_EcCoESdoRead for all CoE reads.
fbCoERead(
	sNetId:= stAX5000_DriveAddress.NetID, 
	nSlaveAddr:= i_nSlaveAddr, 
	nSubIndex:= , 
	nIndex:= , 
	pDstBuf:= , 
	cbBufLen:= , 
	bExecute:= , 
	tTimeout:= T#2S, 
	bBusy=> , 
	bError=> q_xError, 
	nErrId=> q_udiErrorID);

	
// Read the Configured Safety Option For CH-A in The AX5000 Drive
	(*	An advantage OF using the FB_SoERead FUNCTION block Form the MC2_Drive library
		is the NedID is the controller's NetID not the EtherCAT master so it is possible 
		to leave that field with just blank single quotes '' and the TwinCAT system 
		assumes the NetID of the computer for you.
		
		The MC2_Drive library has dependencies on the MC2 library in TwinCAT and Tc3 at this point
		(build 3099.1) doesn't notice the dependancy and add the extra library for you.  You must
		manually add it yourself.
		
			S_0_IDN		: WORD	:= 16#0000;
			S_1_IDN		: WORD	:= 16#1000;
			S_2_IDN		: WORD	:= 16#2000;
			S_3_IDN		: WORD	:= 16#3000;
			S_4_IDN		: WORD	:= 16#4000;
			S_5_IDN		: WORD	:= 16#5000;
			S_6_IDN		: WORD	:= 16#6000;
			S_7_IDN		: WORD	:= 16#7000;
		
			P_0_IDN		: WORD	:= 16#8000;
			P_1_IDN		: WORD	:= 16#9000;
			P_2_IDN		: WORD	:= 16#A000;
			P_3_IDN		: WORD	:= 16#B000;
			P_4_IDN		: WORD	:= 16#C000;
			P_5_IDN		: WORD	:= 16#D000;
			P_6_IDN		: WORD	:= 16#E000;
			P_7_IDN		: WORD	:= 16#F000;
		
		A Few documented SERCOS error codes:
		---------------------------------------
		0x1003 Wrong parameter mode 
		0x1004 Data parameter wrong value size 
		0x1005 False backup parameter type  
		0x1006 Backup list was not IDN 192 
		
		nElement: Element number of the parameter that is to be written. The following values are allowed:
		--------------------------------------------------------------------------------------------------
		Value Description 
		0x01 Data Status 
		0x02 Name (read only) 
		0x04 Attribute 
		0x08 Unit 
		0x10 Minimum 
		0x20 Maximum 
		0x40 Value 
		0x80 Default 		*)
		
fbAX5000_SafetyOptionSoeRead(
	NetId			:= 	stAX5000_DriveAddress.NetID, 
	Idn				:= 	P_0_IDN + 2000, //Requires Tc2_Drive.lib
	Element			:= 	16#40, 
	pDstBuf			:= 	ADR(wSafetyOption), 
	BufLen			:= 	SIZEOF(wSafetyOption), 
	Execute			:= 	TRUE, 
	Timeout			:= 	T#2S, 
	Axis			:= 	iq_stAxisRef, 
	Busy			=> 	, 
	Error			=> 	, 
	AdsErrId		=> 	, 
	SercosErrId		=> 	, 
	Attribute		=> 	) ;
		
IF  wSafetyOption 	= 0  THEN
	q_stAX5805_Diag.sSafetyOption	:= 		'No Safety Option Selected' ;
ELSIF  wSafetyOption	= 1  THEN
	q_stAX5805_Diag.sSafetyOption	:= 		'AX5801 Option Selected' ;
ELSIF  wSafetyOption	= 2  THEN
	q_stAX5805_Diag.sSafetyOption	:= 		'AX5805 Option Selected' ;
ELSE
	q_stAX5805_Diag.sSafetyOption	:= 		'Invalid Option' ;
END_IF

IF NOT fbAX5000_SafetyOptionSoeRead.Error THEN
	q_xError := FALSE;
	q_sErrorDescription := 'No Error';
ELSIF fbAX5000_SafetyOptionSoeRead.Error THEN
	q_xError := TRUE;
	q_sErrorDescription := 'FB_EcCoESdoRead Safety Option';
END_IF

fbAX5000_SafetyOptionSoeRead.Execute := FALSE;

END_FUNCTION_BLOCK

// POUs/HardwareFBs/FB_EL1904Diagnostics
(*=====================================================================
Beckhoff Automation LLC
Copyright 2015 All Rights Reserved
=======================================================================
Description: 
This Program has been supplied by Beckhoff Automation As-Is and is intended only as an example implementation. 
Functionality is not guaranteed. 
This Function Block reads all status and error information known at time of creation of the EL1904.
---------------------------------------------------------------------------------------------------------------
History:
Date		Version			Author							Comment
---------------------------------------------------------------------------------------------------------------
07.08.15	0.10		Jason Erickson				Initial Library Creation.
07.20.15	0.11		Jason Ericskon				Added CoE Read for TwinSAFE Connection State.
08.28.15	0.20		Jason Erickson				Code optimization to eliminate timed data reads.
09.18.15	0.2.1		Jason Erickson				Added new error codes 0x6000 - 0x6002 and Connection Status to the AX5805.
09.24.15	0.2.2		Jason Erickson				Corrected inability to update CASE in FB_EL1904Diagnostics and FB_EL2904Diagnostics.
10.30.15	0.2.3		Jason Erickson				Modified Diagnostic Structure names for ease of use.
*)
FUNCTION_BLOCK FB_EL1904Diagnostics
VAR_INPUT
// EtherCAT Master Device Net ID.
	i_sNetId: STRING;
// Slave Address of the EL1904.
	i_nSlaveAddr: UINT;
// Reset Latched TwinSAFE Error Messages.
	i_xLatchedMessageReset: BOOL;
END_VAR
VAR_OUTPUT
// Structure to hold all EL1904 output information.
	q_stEL1904_Diag: ST_EL1904_DIAGNOSTICS;
// Internal function block errors.
	q_xError: BOOL;
	q_nErrorID: UDINT;
	q_sErrorDescription: STRING;
END_VAR
VAR
// Case Statement.
	iState: INT;
// FB_EcCoESdoRead for all CoE reads.
	fbCoERead: FB_EcCoESdoRead;
// FB_EcCoESdoReadEx for all CoE EX reads.
	fbCoEReadEX: FB_EcCoESdoReadEx;
// Variable to hold data for evaluation, Micro Controller (MC1) 3.3v Nominal Voltage(mV) INPUT of the EL1904.
	wEL1904_MC1_3300mV: WORD;
// Variable to hold data for evaluation, Micro Controller (MC1) 3.3v Nominal Voltage(mV) INPUT of the EL1904
	wEL1904_MC2_3300mV: WORD;
// Variable to hold data for evaluation, Operating Mode of the EL1904.
	wEL1904_OperMode: WORD;
// Variable to hold data for evaluation, Sensor Tests Active/Inactive of the EL1904.
	iEL1904_STActive: INT;
// Variable to hold data for evaluation, Logic of the EL1904 Channels 1 and 2.
	bEL1904_Logic1_2: BYTE;
// Variable to hold data for evaluation, Logic of the EL1904 Channels 3 and 4.
	bEL1904_Logic3_4: BYTE;
// Variable to hold data for evaluation, Sensor Tests Errors of the EL1904.
	wEL1904_SenT: WORD;
// Variable to hold data for evaluation, Error During Two-Channel Evaluation - Diagnostic object 800E:0B of the EL1904.	
			(* The two channels contradict each other (not same value). *)		
	wEL1904_2CHEval: WORD;
// Variable to hold data for evaluation, Error In Safety Mat Operating Mode: Input Pair Disagree - Diagnostic object 800E:0C of the EL1904.	
			(* Input pairs not in the same state (not same value). *)		
	wEL1904_SMiPair: WORD;
// Variable to hold data for evaluation, Error In Safety Mat Operating Mode: External Supply (No test pulses) - Diagnostic object 800E:0D of the EL1904.	
			(* External supply detected (Input channel not getting test pulses). *)	
	wEL1904_SMExtSupply: WORD;
// Variable to hold data for evaluation, Connection State of the EL1904.
	iEL1904_ConnectionState: INT;
END_VAR

CASE iState OF
	0:// Set Parameters to read the Serial Number of the EL1904.			
			fbCoERead.nSubIndex	:= 	16#02;
			fbCoERead.nIndex	:= 	16#F980;
			fbCoERead.pDstBuf	:= 	ADR(q_stEL1904_Diag.dwSerialNumber);
			fbCoERead.cbBufLen	:= 	SIZEOF(q_stEL1904_Diag.dwSerialNumber);
			fbCoERead.bExecute	:= 	TRUE;		
			iState := iState + 10;	
			
	10:// Evaluate read of the Serial Number of the EL1904.			
		IF NOT fbCoERead.bBusy THEN
			fbCoERead.bExecute := FALSE;
			q_sErrorDescription := 'No Error';
			iState := iState + 10;
			IF fbCoERead.bError THEN
				q_sErrorDescription := 'EL1904 Serial Number - Read Error';
			END_IF
		END_IF	
		
	20:// Set Parameters to read the DIP Switch Setting of the EL1904.			
			fbCoERead.nSubIndex	:= 	16#01;
			fbCoERead.nIndex	:= 	16#F980;
			fbCoERead.pDstBuf	:= 	ADR(q_stEL1904_Diag.wDipSwitch);
			fbCoERead.cbBufLen	:= 	SIZEOF(q_stEL1904_Diag.wDipSwitch);
			fbCoERead.bExecute	:= 	TRUE;		
			iState := iState + 10;	
			
	30:// Evaluate read DIP Switch Setting of the EL1904.		
		IF NOT fbCoERead.bBusy THEN
			fbCoERead.bExecute := FALSE;
			q_sErrorDescription := 'No Error';
			iState := iState + 10;
			IF fbCoERead.bError THEN
				q_sErrorDescription := 'EL1904 DIP Switch Setting - Read Error';
			END_IF
		END_IF		

	40:// Set Parameters to read the Hardware Version of the EL1904.			
			fbCoERead.nSubIndex	:= 	0;
			fbCoERead.nIndex	:= 	16#1009;
			fbCoERead.pDstBuf	:= 	ADR(q_stEL1904_Diag.sHwVersion);
			fbCoERead.cbBufLen	:= 	SIZEOF(q_stEL1904_Diag.sHwVersion);
			fbCoERead.bExecute	:= 	TRUE;		
			iState := iState + 10;	
			
	50:// Evaluate read Hardware Version of the EL1904.		
		IF NOT fbCoERead.bBusy THEN
			fbCoERead.bExecute := FALSE;
			q_sErrorDescription := 'No Error';
			iState := iState + 10;
			IF fbCoERead.bError THEN
				q_sErrorDescription := 'EL1904 Hardware Version - Read Error';
			END_IF
		END_IF		

	60:// Set Parameters to read the Software Version (firmware) of the EL1904.			
			fbCoERead.nSubIndex	:= 	0;
			fbCoERead.nIndex	:= 	16#100A;
			fbCoERead.pDstBuf	:= 	ADR(q_stEL1904_Diag.sFwVersion);
			fbCoERead.cbBufLen	:= 	SIZEOF(q_stEL1904_Diag.sFwVersion);
			fbCoERead.bExecute	:= 	TRUE;		
			iState := iState + 10;	
			
	70:// Evaluate read Software Version (firmware) of the EL1904.		
		IF NOT fbCoERead.bBusy THEN
			fbCoERead.bExecute := FALSE;
			q_sErrorDescription := 'No Error';
			iState := iState + 10;
			IF fbCoERead.bError THEN
				q_sErrorDescription := 'EL1904 Software Version - Read Error';
			END_IF
		END_IF		

	80:// Set Parameters to read Micro Controller (MC1) Temperature in DegC of the EL1904.			
			fbCoERead.nSubIndex	:= 	16#01;
			fbCoERead.nIndex	:= 	16#FA80;
			fbCoERead.pDstBuf	:= 	ADR(q_stEL1904_Diag.wMC1Temp);
			fbCoERead.cbBufLen	:= 	SIZEOF(q_stEL1904_Diag.wMC1Temp);
			fbCoERead.bExecute	:= 	TRUE;		
			iState := iState + 10;	
			
	90:// Evaluate read Micro Controller (MC1) Temperature in DegC of the EL1904.		
		IF NOT fbCoERead.bBusy THEN
			fbCoERead.bExecute := FALSE;
			q_sErrorDescription := 'No Error';
			iState := iState + 10;
			IF fbCoERead.bError THEN
				q_sErrorDescription := 'EL1904 MC1 Temp - Read Error';
			END_IF
		END_IF		
		
	100:// Set Parameters to read Micro Controller (MC2) Temperature in DegC of the EL1904.			
			fbCoERead.nSubIndex	:= 	16#02;
			fbCoERead.nIndex	:= 	16#FA80;
			fbCoERead.pDstBuf	:= 	ADR(q_stEL1904_Diag.wMC2Temp);
			fbCoERead.cbBufLen	:= 	SIZEOF(q_stEL1904_Diag.wMC2Temp);
			fbCoERead.bExecute	:= 	TRUE;		
			iState := iState + 10;	
			
	110:// Evaluate read Micro Controller (MC2) Temperature in DegC of the EL1904.		
		IF NOT fbCoERead.bBusy THEN
			fbCoERead.bExecute := FALSE;
			q_sErrorDescription := 'No Error';
			iState := iState + 10;
			IF fbCoERead.bError THEN
				q_sErrorDescription := 'EL1904 MC2 Temp - Read Error';
			END_IF
		END_IF		

	120:// Set Parameters to read Micro Controller (MC1) 3300mv Nominal Voltage INPUT of the EL1904.			
			fbCoERead.nSubIndex	:= 	16#01;
			fbCoERead.nIndex	:= 	16#FA81;
			fbCoERead.pDstBuf	:= 	ADR(wEL1904_MC1_3300mV);
			fbCoERead.cbBufLen	:= 	SIZEOF(wEL1904_MC1_3300mV);
			fbCoERead.bExecute	:= 	TRUE;		
			iState := iState + 10;	
			
	130:// Evaluate read Micro Controller (MC1) 3300mv Nominal Voltage INPUT of the EL1904.		
		IF NOT fbCoERead.bBusy THEN
		 	q_stEL1904_Diag.lrMC1_3300mV :=  WORD_TO_LREAL(wEL1904_MC1_3300mV);
			fbCoERead.bExecute := FALSE;
			q_sErrorDescription := 'No Error';
			iState := iState + 10;
			IF fbCoERead.bError THEN
				q_sErrorDescription := 'EL1904 MC1 3.3v Input - Read Error';
			END_IF
		END_IF	
		
	140:// Set Parameters to read Micro Controller (MC2) 3300mv Nominal Voltage INPUT of the EL1904.			
			fbCoERead.nSubIndex	:= 	16#02;
			fbCoERead.nIndex	:= 	16#FA81;
			fbCoERead.pDstBuf	:= 	ADR(wEL1904_MC2_3300mV);
			fbCoERead.cbBufLen	:= 	SIZEOF(wEL1904_MC2_3300mV);
			fbCoERead.bExecute	:= 	TRUE;		
			iState := iState + 10;	
			
	150:// Evaluate read Micro Controller (MC2) 3300mv Nominal Voltage INPUT of the EL1904.		
		IF NOT fbCoERead.bBusy THEN
		 	q_stEL1904_Diag.lrMC2_3300mV :=  WORD_TO_LREAL(wEL1904_MC2_3300mV);
			fbCoERead.bExecute := FALSE;
			q_sErrorDescription := 'No Error';
			iState := iState + 10;
			IF fbCoERead.bError THEN
				q_sErrorDescription := 'EL1904 MC2 3.3v Input - Read Error';
			END_IF
		END_IF	
	
	160:// Set Parameters to read Operating Mode of the EL1904.			
			fbCoERead.nSubIndex	:= 	16#01;
			fbCoERead.nIndex	:= 	16#8000;
			fbCoERead.pDstBuf	:= 	ADR(wEL1904_OperMode);
			fbCoERead.cbBufLen	:= 	SIZEOF(wEL1904_OperMode);
			fbCoERead.bExecute	:= 	TRUE;		
			iState := iState + 10;	
			
	170:// Evaluate read Operating Mode of the EL1904.		
		IF NOT fbCoERead.bBusy THEN
		 	IF wEL1904_OperMode  =  0 THEN
				q_stEL1904_Diag.sOpMode  :=  'Digital' ;
			ELSIF wEL1904_OperMode  =  1 THEN
				q_stEL1904_Diag.sOpMode  :=  'Standstill Monitoring 1' ;
			ELSIF wEL1904_OperMode  =  2 THEN
				q_stEL1904_Diag.sOpMode  :=  'Standstill Monitoring 2' ;
			ELSE
				q_stEL1904_Diag.sOpMode  :=  'Invalid Mode' ;
			END_IF ;
			fbCoERead.bExecute := FALSE;
			q_sErrorDescription := 'No Error';
			iState := iState + 10;
			IF fbCoERead.bError THEN
				q_sErrorDescription := 'EL1904 Operating Mode - Read Error';
			END_IF
		END_IF	
		
	180:// Set Parameters to read Sensor Tests Active/Inactive of the EL1904.			
			fbCoEReadEX.nSubIndex	:= 	1;
			fbCoEReadEX.nIndex	:= 	16#8001;
			fbCoEReadEX.pDstBuf	:= 	ADR(iEL1904_STActive);
			fbCoEReadEX.cbBufLen	:= 	SIZEOF(iEL1904_STActive);
			fbCoEReadEX.bExecute	:= 	TRUE;		
			iState := iState + 10;	
			
	190:// Evaluate read Sensor Tests Active/Inactive of the EL1904.		
		IF NOT fbCoEReadEX.bBusy THEN
		 	IF NOT iEL1904_STActive.0 THEN
				q_stEL1904_Diag.xSensorTestActive1 := FALSE;
			ELSIF iEL1904_STActive.0 THEN
				q_stEL1904_Diag.xSensorTestActive1 := TRUE;
			END_IF
			
			IF NOT iEL1904_STActive.1 THEN
				q_stEL1904_Diag.xSensorTestActive2 := FALSE;
			ELSIF iEL1904_STActive.1 THEN
				q_stEL1904_Diag.xSensorTestActive2 := TRUE;
			END_IF
			
			IF NOT iEL1904_STActive.2 THEN
				q_stEL1904_Diag.xSensorTestActive3 := FALSE;
			ELSIF iEL1904_STActive.2 THEN
				q_stEL1904_Diag.xSensorTestActive3 := TRUE;
			END_IF
			
			IF NOT iEL1904_STActive.3 THEN
				q_stEL1904_Diag.xSensorTestActive4 := FALSE;
			ELSIF iEL1904_STActive.3 THEN
				q_stEL1904_Diag.xSensorTestActive4 := TRUE;
			END_IF
			fbCoEReadEX.bExecute := FALSE;
			q_sErrorDescription := 'No Error';
			iState := iState + 10;
			IF fbCoEReadEX.bError THEN
				q_sErrorDescription := 'EL1904 Sensor Tests Active/Inactive - Read Error';
			END_IF
		END_IF	
		
	200:// Set Parameters to read Logic of Channels 1 and 2 of the EL1904.			
			fbCoERead.nSubIndex	:= 	1;
			fbCoERead.nIndex	:= 	16#8002;
			fbCoERead.pDstBuf	:= 	ADR(bEL1904_Logic1_2);
			fbCoERead.cbBufLen	:= 	SIZEOF(bEL1904_Logic1_2);
			fbCoERead.bExecute	:= 	TRUE;		
			iState := iState + 10;	
			
	210:// Evaluate read Logic of Channels 1 and 2 of the EL1904.		
		IF NOT fbCoERead.bBusy THEN
		 	IF  bEL1904_Logic1_2  = 0  THEN
				q_stEL1904_Diag.sLogicMode_Ch1Ch2 := 'Single Channel Logic' ;
			ELSIF  bEL1904_Logic1_2  =  1  THEN
				q_stEL1904_Diag.sLogicMode_Ch1Ch2 := 'Asynchronous Repetitive OSSD, Sensor Test Must Be Disabled!' ;
			ELSIF  bEL1904_Logic1_2  =  2  THEN
				q_stEL1904_Diag.sLogicMode_Ch1Ch2 := 'Any Pulse Repetitive OSSD, Sensor Test Must Be Disabled!' ;
			ELSIF  bEL1904_Logic1_2  =  3  THEN
				q_stEL1904_Diag.sLogicMode_Ch1Ch2 := 'Short Cut, No Module Fault' ;
			ELSE
				q_stEL1904_Diag.sLogicMode_Ch1Ch2 := 'Invalid Logic CH1 and CH2' ;
			END_IF ;
			fbCoERead.bExecute := FALSE;
			q_sErrorDescription := 'No Error';
			iState := iState + 10;
			IF fbCoERead.bError THEN
				q_sErrorDescription := 'EL1904 Logic of Channels 1 and 2 - Read Error';
			END_IF
		END_IF	

	220:// Set Parameters to read Logic of Channels 3 and 4 of the EL1904.			
			fbCoERead.nSubIndex	:= 	3;
			fbCoERead.nIndex	:= 	16#8002;
			fbCoERead.pDstBuf	:= 	ADR(bEL1904_Logic3_4);
			fbCoERead.cbBufLen	:= 	SIZEOF(bEL1904_Logic3_4);
			fbCoERead.bExecute	:= 	TRUE;		
			iState := iState + 10;	
			
	230:// Evaluate read Logic of Channels 3 and 4 of the EL1904.		
		IF NOT fbCoERead.bBusy THEN
		 	IF  bEL1904_Logic3_4  = 0  THEN
				q_stEL1904_Diag.sLogicMode_Ch3Ch4  := 'Single Channel Logic' ;
			ELSIF  bEL1904_Logic3_4  = 1  THEN
				q_stEL1904_Diag.sLogicMode_Ch3Ch4  := 'Asynchronous Repetitive OSSD, Sensor Test Must Be Disabled!' ;
			ELSIF  bEL1904_Logic3_4  = 2  THEN
				q_stEL1904_Diag.sLogicMode_Ch3Ch4  := 'Any Pulse Repetitive OSSD, Sensor Test Must Be Disabled!' ;
			ELSIF  bEL1904_Logic3_4  = 3  THEN
				q_stEL1904_Diag.sLogicMode_Ch3Ch4  := 'Short Cut, No Module Fault' ;
			ELSE
				q_stEL1904_Diag.sLogicMode_Ch3Ch4  := 'Invalid Logic CH3 and CH4' ;
			END_IF ;		
			fbCoERead.bExecute := FALSE;
			q_sErrorDescription := 'No Error';
			iState := iState + 10;
			IF fbCoERead.bError THEN
				q_sErrorDescription := 'EL1904 Logic of Channels 3 and 4 - Read Error';
			END_IF
		END_IF	

(**************************************ALARMS**************************************)
(**************************************ALARMS**************************************)
(**************************************ALARMS**************************************)	
	240:// Set Parameters to read Sensor Test Error of the EL1904.			
			fbCoERead.nSubIndex	:= 	16#0A;
			fbCoERead.nIndex	:= 	16#800E;
			fbCoERead.pDstBuf	:= 	ADR(wEL1904_SenT);
			fbCoERead.cbBufLen	:= 	SIZEOF(wEL1904_SenT);
			fbCoERead.bExecute	:= 	TRUE;		
			iState := iState + 10;	
			
	250:// Evaluate read Sensor Test Error of the EL1904.		
		IF NOT fbCoERead.bBusy THEN
		 	(* These errors may only be present temporarily so they need to be latched and then cleared
				to be properly noted by the operator. *)
			IF wEL1904_SenT.0 OR wEL1904_SenT.1 OR wEL1904_SenT.2 OR wEL1904_SenT.3 THEN
				q_stEL1904_Diag.xSensorTest1_Error 	:= 	wEL1904_SenT.0;
				q_stEL1904_Diag.xSensorTest2_Error 	:= 	wEL1904_SenT.1;
				q_stEL1904_Diag.xSensorTest3_Error 	:= 	wEL1904_SenT.2;
				q_stEL1904_Diag.xSensorTest4_Error 	:=  wEL1904_SenT.3;
			ELSIF i_xLatchedMessageReset THEN
				q_stEL1904_Diag.xSensorTest1_Error	:= FALSE;
				q_stEL1904_Diag.xSensorTest2_Error	:= FALSE;
				q_stEL1904_Diag.xSensorTest3_Error	:= FALSE;
				q_stEL1904_Diag.xSensorTest4_Error	:= FALSE;
			END_IF
			fbCoERead.bExecute := FALSE;
			q_sErrorDescription := 'No Error';
			iState := iState + 10;
			IF fbCoERead.bError THEN
				q_sErrorDescription := 'EL1904 Sensor Test Error - Read Error';
			END_IF
		END_IF	
		
	260:// Set Parameters to read Error During Two-Channel Evaluation - Diagnostic object 800E:0B of the EL1904.	
			(* The two channels contradict each other (not same value). *)		
			fbCoERead.nSubIndex	:= 	16#0B;
			fbCoERead.nIndex	:= 	16#800E;
			fbCoERead.pDstBuf	:= 	ADR(wEL1904_2CHEval);
			fbCoERead.cbBufLen	:= 	SIZEOF(wEL1904_2CHEval);
			fbCoERead.bExecute	:= 	TRUE;		
			iState := iState + 10;	
			
	270:// Evaluate read Error During Two-Channel Evaluation - Diagnostic object 800E:0B of the EL1904.	
			(* The two channels contradict each other (not same value). *)			
		IF NOT fbCoERead.bBusy THEN
		 	(* These errors may only be present temporarily so they need to be latched and then cleared
				to be properly noted by the operator. *)
			IF wEL1904_2CHEval.0 OR wEL1904_2CHEval.1 THEN
				q_stEL1904_Diag.x2ChanEvalError_Pair1	 :=  wEL1904_2CHEval.0;
				q_stEL1904_Diag.x2ChanEvalError_Pair2	 :=  wEL1904_2CHEval.1;
			ELSIF i_xLatchedMessageReset THEN
				q_stEL1904_Diag.x2ChanEvalError_Pair1	:= FALSE;
				q_stEL1904_Diag.x2ChanEvalError_Pair2	:= FALSE;
			END_IF	
			fbCoERead.bExecute := FALSE;
			q_sErrorDescription := 'No Error';
			iState := iState + 10;
			IF fbCoERead.bError THEN
				q_sErrorDescription := 'EL1904 Error During Two-Channel Evaluation - Read Error';
			END_IF
		END_IF	

	280:// Set Parameters to read Error In Safety Mat Operating Mode: Input Pair Disagree - Diagnostic object 800E:0C of the EL1904.	
			(* Input pairs not in the same state (not same value). *)		
			fbCoERead.nSubIndex	:= 	16#0C;
			fbCoERead.nIndex	:= 	16#800E;
			fbCoERead.pDstBuf	:= 	ADR(wEL1904_SMiPair);
			fbCoERead.cbBufLen	:= 	SIZEOF(wEL1904_SMiPair);
			fbCoERead.bExecute	:= 	TRUE;		
			iState := iState + 10;	
			
	290:// Evaluate read Error In Safety Mat Operating Mode: Input Pair Disagree - Diagnostic object 800E:0C of the EL1904.	
			(* Input pairs not in the same state (not same value). *)			
		IF NOT fbCoERead.bBusy THEN
		 	(* These errors may only be present temporarily so they need to be latched and then cleared
				to be properly noted by the operator. *)
			IF (wEL1904_SMiPair.0 AND wEL1904_SMiPair.1) OR (wEL1904_SMiPair.2 AND wEL1904_SMiPair.3) THEN
				q_stEL1904_Diag.xSafeMatError_Pair1	 :=  (wEL1904_SMiPair.0  AND  wEL1904_SMiPair.1);
				q_stEL1904_Diag.xSafeMatError_Pair2	 :=  (wEL1904_SMiPair.2  AND  wEL1904_SMiPair.3);
			ELSIF i_xLatchedMessageReset THEN
				q_stEL1904_Diag.xSafeMatError_Pair1	:= FALSE;
				q_stEL1904_Diag.xSafeMatError_Pair2	:= FALSE;
			END_IF
			fbCoERead.bExecute := FALSE;
			q_sErrorDescription := 'No Error';
			iState := iState + 10;
			IF fbCoERead.bError THEN
				q_sErrorDescription := 'EL1904 Error In Safety Mat Operating Mode: Input Pair Disagree - Read Error';
			END_IF
		END_IF	

	300:// Set Parameters to read Error In Safety Mat Operating Mode: External Supply (No test pulses) - Diagnostic object 800E:0D of the EL1904.	
			(* External supply detected (Input channel not getting test pulses). *)		
			fbCoERead.nSubIndex	:= 	16#0D;
			fbCoERead.nIndex	:= 	16#800E;
			fbCoERead.pDstBuf	:= 	ADR(wEL1904_SMExtSupply);
			fbCoERead.cbBufLen	:= 	SIZEOF(wEL1904_SMExtSupply);
			fbCoERead.bExecute	:= 	TRUE;		
			iState := iState + 10;	
			
	310:// Evaluate read Error In Safety Mat Operating Mode: External Supply (No test pulses) - Diagnostic object 800E:0D of the EL1904.	
			(* External supply detected (Input channel not getting test pulses). *)			
		IF NOT fbCoERead.bBusy THEN
		 	(* These errors may only be present temporarily so they need to be latched and then cleared
				to be properly noted by the operator. *)
			IF wEL1904_SMExtSupply > 0  THEN
				q_stEL1904_Diag.xSafeMatExternalSupplyErrorCh1  := 	wEL1904_SMExtSupply.0;
				q_stEL1904_Diag.xSafeMatExternalSupplyErrorCh2  := 	wEL1904_SMExtSupply.2;
				q_stEL1904_Diag.xSafeMatExternalSupplyErrorCh3  := 	wEL1904_SMExtSupply.3;
				q_stEL1904_Diag.xSafeMatExternalSupplyErrorCh4  := 	wEL1904_SMExtSupply.4;
			ELSIF i_xLatchedMessageReset THEN
				q_stEL1904_Diag.xSafeMatExternalSupplyErrorCh1	:= FALSE;
				q_stEL1904_Diag.xSafeMatExternalSupplyErrorCh2	:= FALSE;
				q_stEL1904_Diag.xSafeMatExternalSupplyErrorCh3	:= FALSE;
				q_stEL1904_Diag.xSafeMatExternalSupplyErrorCh4	:= FALSE;
			END_IF
			fbCoERead.bExecute := FALSE;
			q_sErrorDescription := 'No Error';
			iState := iState + 10;
			IF fbCoERead.bError THEN
				q_sErrorDescription := 'EL1904 Error In Safety Mat Operating Mode: External Supply - Read Error';
			END_IF
		END_IF	

	320:// Set Parameters to read Connection State of the EL1904.	
			fbCoERead.nSubIndex	:= 	1;
			fbCoERead.nIndex	:= 	16#A000;
			fbCoERead.pDstBuf	:= 	ADR(iEL1904_ConnectionState);
			fbCoERead.cbBufLen	:= 	SIZEOF(iEL1904_ConnectionState);
			fbCoERead.bExecute	:= 	TRUE;		
			iState := iState + 10;	
			
	330:// Evaluate read Connection State of the EL1904.	
		IF NOT fbCoERead.bBusy THEN
		 	(* These errors may only be present temporarily so they need to be latched and then cleared
				to be properly noted by the operator. *)
			IF iEL1904_ConnectionState = 0 THEN
				q_stEL1904_Diag.sConnectionState := 'Reset State';
			ELSIF iEL1904_ConnectionState = 1 THEN
				q_stEL1904_Diag.sConnectionState := 'Session State';
			ELSIF iEL1904_ConnectionState = 2 THEN
				q_stEL1904_Diag.sConnectionState := 'Connection State';
			ELSIF iEL1904_ConnectionState = 3 THEN
				q_stEL1904_Diag.sConnectionState := 'Parameter State';
			ELSIF iEL1904_ConnectionState = 4 THEN
				q_stEL1904_Diag.sConnectionState := 'Data State';
			ELSIF iEL1904_ConnectionState = 5 THEN
				q_stEL1904_Diag.sConnectionState := 'Failsafe State';
			ELSE
				q_stEL1904_Diag.sConnectionState := 'Undefined State';
			END_IF
			fbCoERead.bExecute := FALSE;
			q_sErrorDescription := 'No Error';
			iState := 0;
			IF fbCoERead.bError THEN
				q_sErrorDescription := 'EL1904 Connection State - Read Error';
			END_IF
		END_IF	
END_CASE

// FB_EcCoESdoRead for all CoE reads.
fbCoERead(
	sNetId:= i_sNetId, 
	nSlaveAddr:= i_nSlaveAddr, 
	nSubIndex:= , 
	nIndex:= , 
	pDstBuf:= , 
	cbBufLen:= , 
	bExecute:= , 
	tTimeout:= T#2S, 
	bBusy=> , 
	bError=> q_xError, 
	nErrId=> q_nErrorID);

// FB_EcCoESdoReadEx for all CoE EX reads.
fbCoEReadEX(
	sNetId:= i_sNetId, 
	nSlaveAddr:= i_nSlaveAddr, 
	nSubIndex:= , 
	nIndex:= , 
	pDstBuf:= , 
	cbBufLen:= , 
	bExecute:= , 
	tTimeout:= T#2S, 
	bCompleteAccess:= TRUE, 
	bBusy=> , 
	bError=> q_xError, 
	nErrId=> q_nErrorID);

// If any of above errors exist set q_stEL1904_Diag.xEL1904Error TRUE.
IF NOT q_stEL1904_Diag.x2ChanEvalError_Pair1 OR
	q_stEL1904_Diag.x2ChanEvalError_Pair2 OR
	q_stEL1904_Diag.xSafeMatError_Pair1 OR
	q_stEL1904_Diag.xSafeMatError_Pair2 OR
	q_stEL1904_Diag.xSafeMatExternalSupplyErrorCh1 OR
	q_stEL1904_Diag.xSafeMatExternalSupplyErrorCh2 OR
	q_stEL1904_Diag.xSafeMatExternalSupplyErrorCh3 OR
	q_stEL1904_Diag.xSafeMatExternalSupplyErrorCh4 OR
	q_stEL1904_Diag.xSensorTest1_Error OR
	q_stEL1904_Diag.xSensorTest2_Error OR
	q_stEL1904_Diag.xSensorTest3_Error OR
	q_stEL1904_Diag.xSensorTest4_Error THEN
		q_stEL1904_Diag.xEL1904Error := FALSE;
ELSIF q_stEL1904_Diag.x2ChanEvalError_Pair1 OR
	q_stEL1904_Diag.x2ChanEvalError_Pair2 OR
	q_stEL1904_Diag.xSafeMatError_Pair1 OR
	q_stEL1904_Diag.xSafeMatError_Pair2 OR
	q_stEL1904_Diag.xSafeMatExternalSupplyErrorCh1 OR
	q_stEL1904_Diag.xSafeMatExternalSupplyErrorCh2 OR
	q_stEL1904_Diag.xSafeMatExternalSupplyErrorCh3 OR
	q_stEL1904_Diag.xSafeMatExternalSupplyErrorCh4 OR
	q_stEL1904_Diag.xSensorTest1_Error OR
	q_stEL1904_Diag.xSensorTest2_Error OR
	q_stEL1904_Diag.xSensorTest3_Error OR
	q_stEL1904_Diag.xSensorTest4_Error THEN
		q_stEL1904_Diag.xEL1904Error := TRUE;
END_IF

END_FUNCTION_BLOCK

// POUs/HardwareFBs/FB_EL2904Diagnostics
(*=====================================================================
Beckhoff Automation LLC
Copyright 2015 All Rights Reserved
=======================================================================
Description: 
This Program has been supplied by Beckhoff Automation As-Is and is intended only as an example implementation. 
Functionality is not guaranteed. 
This Function Block reads all status and error information known at time of creation of the EL2904.
---------------------------------------------------------------------------------------------------------------
History:
Date		Version			Author							Comment
---------------------------------------------------------------------------------------------------------------
07.08.15	0.10		Jason Erickson				Initial Library Creation.
07.20.15	0.11		Jason Ericskon				Added CoE Read for TwinSAFE Connection State.
08.28.15	0.20		Jason Erickson				Code optimization to eliminate timed data reads.
09.18.15	0.2.1		Jason Erickson				Added new error codes 0x6000 - 0x6002 and Connection Status to the AX5805.
09.24.15	0.2.2		Jason Erickson				Corrected inability to update CASE in FB_EL1904Diagnostics and FB_EL2904Diagnostics.
10.30.15	0.2.3		Jason Erickson				Modified Diagnostic Structure names for ease of use.
*)
FUNCTION_BLOCK FB_EL2904Diagnostics
VAR_INPUT
// EtherCAT Master Device Net ID.
	i_sNetId: STRING;
// Slave Address of the EL2904.
	i_nSlaveAddr: UINT;
// Input to reset Latched TwinSAFE Error Messages.
	i_xLatchedMessageReset: BOOL;
END_VAR
VAR_OUTPUT
// Structure to hold all EL2904 output information.
	q_stEL2904_Diag: ST_EL2904_DIAGNOSTICS;
// Internal function block errors.
	q_xError: BOOL;
	q_nErrorID: UDINT;
	q_sErrorDescription: STRING;
END_VAR
VAR
// Case Statement.
	iState: INT;
// FB_EcCoESdoRead for all CoE reads.
	fbCoERead: FB_EcCoESdoRead;
// Variable to hold data for evaluation, Micro Controller (MC1) 3.3v Nominal Voltage(mV) INPUT of the EL2904.
	wEL2904_MC1_3300mV: WORD;
// Variable to hold data for evaluation, Micro Controller (MC2) 3.3v Nominal Voltage(mV) INPUT of the EL2904.
	wEL2904_MC2_3300mV: WORD;
// Variable to hold data for evaluation, Standard Output Active/Inactive of the EL2904.
		(* Standard outputs can be used to directly Enable/Disable a TwinSAFE output
			if this feature is ACTIVE (Not to Turn it ON/OFF, Allow it or not to turn ON!!! *)
	bEL2904_StandardOuts: BYTE;
// Variable to hold data for evaluation, Current Measurement Active/Inactive of the EL2904.		
		(* Used to determine TwinSAFE output load current issues. *)	
	bEL2904_CurrMeas: BYTE;
// Variable to hold data for evaluation, Test Pulses Active/Inactive of the EL2904.
		(* Used to determine TwinSAFE output wiring is correct. *)	
	bEL2904_TestP: BYTE;
// Variable to hold data for evaluation, Output Error Acknowledge Active/Inactive of the EL2904.
		(* Used to reset TwinSAFE output errors instead of forcing a cycle power for a TwinSAFE output error. *)	
	bEL2904_ErrAck: BYTE;
// Variable to hold data for evaluation, Error At The Output of the EL2904.
		(* Bit0-3 is External supply or cross-circuit Error,
			Bit4-7 is Open Load, Current Below 20mA, or Current Above Maximum Value of 500mA. *)
	wEL2904_OutErr: WORD;
// Variable to hold data for evaluation, Power Rail Supply Error of the EL2904 - Field Potential Too High or Too Low
		(*Documentation says this is in 800E:0D but testing shows it's in 800E:0A
			Value = 0x1101 when voltage is below 17.4 v
			Value = 0x1110 when voltage is above 20.8v. *)	
	wEL2904_SupplyErr: WORD;
// Variable to hold data for evaluation, Internal Chip Temperature Error of the EL2904.
		(* There are two temperature sensors inside each Microcontroller and another on the Output Circuit Board. *)	
	wEL2904_TempErr: WORD;
// Variable to hold data for evaluation, Connection State of the EL2904.
	iEL2904_ConnectionState: INT;
END_VAR

CASE iState OF
	0:// Set Parameters to read the Serial Number of the EL2904.			
			fbCoERead.nSubIndex	:= 	16#02;
			fbCoERead.nIndex	:= 	16#F980;
			fbCoERead.pDstBuf	:= 	ADR(q_stEL2904_Diag.dwSerialNumber);
			fbCoERead.cbBufLen	:= 	SIZEOF(q_stEL2904_Diag.dwSerialNumber);
			fbCoERead.bExecute	:= 	TRUE;		
			iState := iState + 10;	
			
	10:// Evaluate read of the Serial Number of the EL2904.			
		IF NOT fbCoERead.bBusy THEN
			fbCoERead.bExecute := FALSE;
			q_sErrorDescription := 'No Error';
			iState := iState + 10;
			IF fbCoERead.bError THEN
				q_sErrorDescription := 'EL2904 Serial Number - Read Error';
			END_IF
		END_IF		
		
	20:// Set Parameters to read the DIP Switch Setting of the EL2904.			
			fbCoERead.nSubIndex	:= 	16#01;
			fbCoERead.nIndex	:= 	16#F980;
			fbCoERead.pDstBuf	:= 	ADR(q_stEL2904_Diag.wDipSwitch);
			fbCoERead.cbBufLen	:= 	SIZEOF(q_stEL2904_Diag.wDipSwitch);
			fbCoERead.bExecute	:= 	TRUE;		
			iState := iState + 10;	
			
	30:// Evaluate read of the DIP Switch Setting of the EL2904.			
		IF NOT fbCoERead.bBusy THEN
			fbCoERead.bExecute := FALSE;
			q_sErrorDescription := 'No Error';
			iState := iState + 10;
			IF fbCoERead.bError THEN
				q_sErrorDescription := 'EL2904 DIP Switch Setting - Read Error';
			END_IF
		END_IF		
		
	40:// Set Parameters to read the Hardware Version of the EL2904.			
			fbCoERead.nSubIndex	:= 	0;
			fbCoERead.nIndex	:= 	16#1009;
			fbCoERead.pDstBuf	:= 	ADR(q_stEL2904_Diag.sHwVersion);
			fbCoERead.cbBufLen	:= 	SIZEOF(q_stEL2904_Diag.sHwVersion);
			fbCoERead.bExecute	:= 	TRUE;		
			iState := iState + 10;	
			
	50:// Evaluate read of the Hardware Version of the EL2904.			
		IF NOT fbCoERead.bBusy THEN
			fbCoERead.bExecute := FALSE;
			q_sErrorDescription := 'No Error';
			iState := iState + 10;
			IF fbCoERead.bError THEN
				q_sErrorDescription := 'EL2904 Hardware Version - Read Error';
			END_IF
		END_IF			
	
	60:// Set Parameters to read the Software Version (firmware) of the EL2904.			
		fbCoERead.nSubIndex	:= 	0;
		fbCoERead.nIndex	:= 	16#100A;
		fbCoERead.pDstBuf	:= 	ADR(q_stEL2904_Diag.sFwVersion);
		fbCoERead.cbBufLen	:= 	SIZEOF(q_stEL2904_Diag.sFwVersion);
		fbCoERead.bExecute	:= 	TRUE;		
		iState := iState + 10;	
			
	70:// Evaluate read of the Software Version (firmware) of the EL2904.			
		IF NOT fbCoERead.bBusy THEN
			fbCoERead.bExecute := FALSE;
			q_sErrorDescription := 'No Error';
			iState := iState + 10;
			IF fbCoERead.bError THEN
				q_sErrorDescription := 'EL2904 Software Version (firmware) - Read Error';
			END_IF
		END_IF	
	
	80:// Set Parameters to read Micro Controller (MC1) Temperature in DegC of the EL2904.			
		fbCoERead.nSubIndex	:= 	16#01;
		fbCoERead.nIndex	:= 	16#FA80;
		fbCoERead.pDstBuf	:= 	ADR(q_stEL2904_Diag.wMC1Temp);
		fbCoERead.cbBufLen	:= 	SIZEOF(q_stEL2904_Diag.wMC1Temp);
		fbCoERead.bExecute	:= 	TRUE;		
		iState := iState + 10;	
			
	90:// Evaluate read Micro Controller (MC1) Temperature in DegC of the EL2904.			
		IF NOT fbCoERead.bBusy THEN
			fbCoERead.bExecute := FALSE;
			q_sErrorDescription := 'No Error';
			iState := iState + 10;
			IF fbCoERead.bError THEN
				q_sErrorDescription := 'EL2904 MC1 Temp - Read Error';
			END_IF
		END_IF	
		
	100:// Set Parameters to read Micro Controller (MC2) Temperature in DegC of the EL2904.			
		fbCoERead.nSubIndex	:= 	16#02;
		fbCoERead.nIndex	:= 	16#FA80;
		fbCoERead.pDstBuf	:= 	ADR(q_stEL2904_Diag.wMC2Temp);
		fbCoERead.cbBufLen	:= 	SIZEOF(q_stEL2904_Diag.wMC2Temp);
		fbCoERead.bExecute	:= 	TRUE;		
		iState := iState + 10;	
			
	110:// Evaluate read Micro Controller (MC2) Temperature in DegC of the EL2904.			
		IF NOT fbCoERead.bBusy THEN
			fbCoERead.bExecute := FALSE;
			q_sErrorDescription := 'No Error';
			iState := iState + 10;
			IF fbCoERead.bError THEN
				q_sErrorDescription := 'EL2904 MC2 Temp - Read Error';
			END_IF
		END_IF	

	120:// Set Parameters to read Micro Controller (MC1) 3300mv Nominal Voltage INPUT of the EL2904.			
		fbCoERead.nSubIndex	:= 	16#01;
		fbCoERead.nIndex	:= 	16#FA81;
		fbCoERead.pDstBuf	:= 	ADR(wEL2904_MC1_3300mV);
		fbCoERead.cbBufLen	:= 	SIZEOF(wEL2904_MC1_3300mV);
		fbCoERead.bExecute	:= 	TRUE;		
		iState := iState + 10;	
			
	130:// Evaluate read Micro Controller (MC1) 3300mv Nominal Voltage INPUT of the EL2904.			
		IF NOT fbCoERead.bBusy THEN
			q_stEL2904_Diag.lrMC1_3300mV  :=  WORD_TO_LREAL(wEL2904_MC1_3300mV);
			fbCoERead.bExecute := FALSE;
			q_sErrorDescription := 'No Error';
			iState := iState + 10;
			IF fbCoERead.bError THEN
				q_sErrorDescription := 'EL2904 MC1 3.3v Input - Read Error';
			END_IF
		END_IF	

	140:// Set Parameters to read Micro Controller (MC2) 3300mv Nominal Voltage INPUT of the EL2904.			
		fbCoERead.nSubIndex	:= 	16#02;
		fbCoERead.nIndex	:= 	16#FA81;
		fbCoERead.pDstBuf	:= 	ADR(wEL2904_MC2_3300mV);
		fbCoERead.cbBufLen	:= 	SIZEOF(wEL2904_MC2_3300mV);
		fbCoERead.bExecute	:= 	TRUE;		
		iState := iState + 10;	
			
	150:// Evaluate read Micro Controller (MC2) 3300mv Nominal Voltage INPUT of the EL2904.			
		IF NOT fbCoERead.bBusy THEN
			q_stEL2904_Diag.lrMC2_3300mV  :=  WORD_TO_LREAL(wEL2904_MC2_3300mV);
			fbCoERead.bExecute := FALSE;
			q_sErrorDescription := 'No Error';
			iState := iState + 10;
			IF fbCoERead.bError THEN
				q_sErrorDescription := 'EL2904 MC2 3.3v Input - Read Error';
			END_IF
		END_IF	

	160:// Standard Output Active/Inactive of the EL2904.
		(* Standard outputs can be used to directly Enable/Disable a TwinSAFE output
			if this feature is ACTIVE (Not to Turn it ON/OFF, Allow it or not to turn ON!!! *)			
		fbCoERead.nSubIndex	:= 	16#01;
		fbCoERead.nIndex	:= 	16#8000;
		fbCoERead.pDstBuf	:= 	ADR(bEL2904_StandardOuts);
		fbCoERead.cbBufLen	:= 	SIZEOF(bEL2904_StandardOuts);
		fbCoERead.bExecute	:= 	TRUE;		
		iState := iState + 10;	
			
	170:// Standard Output Active/Inactive of the EL2904.
		(* Standard outputs can be used to directly Enable/Disable a TwinSAFE output
			if this feature is ACTIVE (Not to Turn it ON/OFF, Allow it or not to turn ON!!! *)				
		IF NOT fbCoERead.bBusy THEN
			q_stEL2904_Diag.xStandardOutputActive  :=  bEL2904_StandardOuts.0 ;
			fbCoERead.bExecute := FALSE;
			q_sErrorDescription := 'No Error';
			iState := iState + 10;
			IF fbCoERead.bError THEN
				q_sErrorDescription := 'EL2904 Standard Output Active/Inactive - Read Error';
			END_IF
		END_IF	

	180:// Set Parameters to read Current Measurement Active/Inactive of the EL2904.		
		(* Used to determine TwinSAFE output load current issues. *)			
		fbCoERead.nSubIndex	:= 	16#02;
		fbCoERead.nIndex	:= 	16#8000;
		fbCoERead.pDstBuf	:= 	ADR(bEL2904_CurrMeas);
		fbCoERead.cbBufLen	:= 	SIZEOF(bEL2904_CurrMeas);
		fbCoERead.bExecute	:= 	TRUE;		
		iState := iState + 10;	
			
	190:// Evaluate read Current Measurement Active/Inactive of the EL2904.		
		(* Used to determine TwinSAFE output load current issues. *)				
		IF NOT fbCoERead.bBusy THEN
			q_stEL2904_Diag.xCurrentMeasureActive  :=  bEL2904_CurrMeas.0 ;
			fbCoERead.bExecute := FALSE;
			q_sErrorDescription := 'No Error';
			iState := iState + 10;
			IF fbCoERead.bError THEN
				q_sErrorDescription := 'EL2904 Current Measurement Active/Inactive - Read Error';
			END_IF
		END_IF	
	
	200:// Set Parameters to read Test Pulses Active/Inactive of the EL2904.
		(* Used to determine TwinSAFE output wiring is correct. *)			
		fbCoERead.nSubIndex	:= 	16#03;
		fbCoERead.nIndex	:= 	16#8000;
		fbCoERead.pDstBuf	:= 	ADR(bEL2904_TestP);
		fbCoERead.cbBufLen	:= 	SIZEOF(bEL2904_TestP);
		fbCoERead.bExecute	:= 	TRUE;		
		iState := iState + 10;	
			
	210:// Evaluate read Test Pulses Active/Inactive of the EL2904.		
		(* Used to determine TwinSAFE output wiring is correct. *)				
		IF NOT fbCoERead.bBusy THEN
			q_stEL2904_Diag.xTestPulsesActive  :=  bEL2904_TestP.0 ;
			fbCoERead.bExecute := FALSE;
			q_sErrorDescription := 'No Error';
			iState := iState + 10;
			IF fbCoERead.bError THEN
				q_sErrorDescription := 'EL2904 Test Pulses Active/Inactive - Read Error';
			END_IF
		END_IF		

	220://Set Parameters to read Output Error Acknowledge Active/Inactive of the EL2904.
		(* Used to reset TwinSAFE output errors instead of forcing a cycle power for a TwinSAFE output error. *)		
		fbCoERead.nSubIndex	:= 	16#04;
		fbCoERead.nIndex	:= 	16#8000;
		fbCoERead.pDstBuf	:= 	ADR(bEL2904_ErrAck);
		fbCoERead.cbBufLen	:= 	SIZEOF(bEL2904_ErrAck);
		fbCoERead.bExecute	:= 	TRUE;		
		iState := iState + 10;	
			
	230:// Evaluate read Output Error Acknowledge Active/Inactive of the EL2904.
		(* Used to reset TwinSAFE output errors instead of forcing a cycle power for a TwinSAFE output error. *)				
		IF NOT fbCoERead.bBusy THEN
			q_stEL2904_Diag.xOutputErrAckActive  :=  bEL2904_ErrAck.0 ;
			fbCoERead.bExecute := FALSE;
			q_sErrorDescription := 'No Error';
			iState := iState + 10;
			IF fbCoERead.bError THEN
				q_sErrorDescription := 'EL2904 Output Error Acknowledge Active/Inactive - Read Error';
			END_IF
		END_IF	

	240://Set Parameters to read Error At The Output of the EL2904.
		(* Bit0-3 is External supply or cross-circuit Error,
			Bit4-7 is Open Load, Current Below 20mA, or Current Above Maximum Value of 500mA. *)
		fbCoERead.nSubIndex	:= 	16#0C;
		fbCoERead.nIndex	:= 	16#800E;
		fbCoERead.pDstBuf	:= 	ADR(wEL2904_OutErr);
		fbCoERead.cbBufLen	:= 	SIZEOF(wEL2904_OutErr);
		fbCoERead.bExecute	:= 	TRUE;		
		iState := iState + 10;	
			
	250:// Evaluate read Output Error Acknowledge Active/Inactive of the EL2904.
		(* Used to reset TwinSAFE output errors instead of forcing a cycle power for a TwinSAFE output error. *)				
		IF NOT fbCoERead.bBusy THEN
			(* These errors may only be present temporarily so they need to be latched and then cleared
				to be properly noted by the operator. *)
		IF wEL2904_OutErr > 0 THEN
			q_stEL2904_Diag.xExternalSupplyOrCrossCircuitError1	:= 		wEL2904_OutErr.0 ;
			q_stEL2904_Diag.xExternalSupplyOrCrossCircuitError2	:= 		wEL2904_OutErr.1 ;
			q_stEL2904_Diag.xExternalSupplyOrCrossCircuitError3	:= 		wEL2904_OutErr.2 ;
			q_stEL2904_Diag.xExternalSupplyOrCrossCircuitError4	:= 		wEL2904_OutErr.3 ;
			q_stEL2904_Diag.xLoadError1		:= 		wEL2904_OutErr.4 ;
			q_stEL2904_Diag.xLoadError2		:= 		wEL2904_OutErr.5 ;
			q_stEL2904_Diag.xLoadError3		:= 		wEL2904_OutErr.6 ;
			q_stEL2904_Diag.xLoadError4		:= 		wEL2904_OutErr.7 ;
		ELSIF i_xLatchedMessageReset THEN
			q_stEL2904_Diag.xExternalSupplyOrCrossCircuitError1 := FALSE;
			q_stEL2904_Diag.xExternalSupplyOrCrossCircuitError2 := FALSE;
			q_stEL2904_Diag.xExternalSupplyOrCrossCircuitError3 := FALSE;
			q_stEL2904_Diag.xExternalSupplyOrCrossCircuitError4 := FALSE;
			q_stEL2904_Diag.xLoadError1 := FALSE;
			q_stEL2904_Diag.xLoadError2 := FALSE;
			q_stEL2904_Diag.xLoadError3 := FALSE;
			q_stEL2904_Diag.xLoadError4 := FALSE;
		END_IF
			fbCoERead.bExecute := FALSE;
			q_sErrorDescription := 'No Error';
			iState := iState + 10;
			IF fbCoERead.bError THEN
				q_sErrorDescription := 'EL2904 Output Error Acknowledge Active/Inactive - Read Error';
			END_IF
		END_IF	
	
	260://Set Parameters to read Power Rail Supply Error of the EL2904 - Field Potential Too High or Too Low
		(*Documentation says this is in 800E:0D but testing shows it's in 800E:0A
			Value = 0x1101 when voltage is below 17.4 v
			Value = 0x1110 when voltage is above 20.8v. *)	
		fbCoERead.nSubIndex	:= 	16#0A;
		fbCoERead.nIndex	:= 	16#800E;
		fbCoERead.pDstBuf	:= 	ADR(wEL2904_SupplyErr);
		fbCoERead.cbBufLen	:= 	SIZEOF(wEL2904_SupplyErr);
		fbCoERead.bExecute	:= 	TRUE;		
		iState := iState + 10;	
			
	270:// Evaluate read Power Rail Supply Error of the EL2904 - Field Potential Too High or Too Low
		(*Documentation says this is in 800E:0D but testing shows it's in 800E:0A
			Value = 0x1101 when voltage is below 17.4 v
			Value = 0x1110 when voltage is above 20.8v. *)				
		IF NOT fbCoERead.bBusy THEN
			(* These errors may only be present temporarily so they need to be latched and then cleared
				to be properly noted BY the operator. *)
			IF wEL2904_SupplyErr.0 OR wEL2904_SupplyErr.1 OR wEL2904_SupplyErr.2 OR wEL2904_SupplyErr.3 THEN
				q_stEL2904_Diag.xPowerRailSupplyVoltHighError	:= 	(NOT wEL2904_SupplyErr.0 AND wEL2904_SupplyErr.1 AND wEL2904_SupplyErr.2 AND wEL2904_SupplyErr.3);
				q_stEL2904_Diag.xPowerRailSupplyVoltLowError	:= 	(wEL2904_SupplyErr.0 AND wEL2904_SupplyErr.1 AND NOT wEL2904_SupplyErr.2 AND wEL2904_SupplyErr.3);
			ELSIF i_xLatchedMessageReset THEN
				q_stEL2904_Diag.xPowerRailSupplyVoltHighError := FALSE;
				q_stEL2904_Diag.xPowerRailSupplyVoltLowError := FALSE;
			END_IF
			fbCoERead.bExecute := FALSE;
			q_sErrorDescription := 'No Error';
			iState := iState + 10;
			IF fbCoERead.bError THEN
				q_sErrorDescription := 'EL2904 Power Rail Supply Error - Read Error';
			END_IF
		END_IF	
								
	280://Set Parameters to read Internal Chip Temperature Error of the EL2904.
		(* There are two temperature sensors inside each Microcontroller and another on the Output Circuit Board. *)			
		fbCoERead.nSubIndex	:= 	16#0E;
		fbCoERead.nIndex	:= 	16#800E;
		fbCoERead.pDstBuf	:= 	ADR(wEL2904_TempErr);
		fbCoERead.cbBufLen	:= 	SIZEOF(wEL2904_TempErr);
		fbCoERead.bExecute	:= 	TRUE;		
		iState := iState + 10;	
			
	290:// Evaluate read Internal Chip Temperature Error of the EL2904.
		(* There are two temperature sensors inside each Microcontroller and another on the Output Circuit Board. *)			
		IF NOT fbCoERead.bBusy THEN
			IF wEL2904_TempErr > 0 THEN
				q_stEL2904_Diag.xOverTempMC1			:= 		wEL2904_TempErr.0;
				q_stEL2904_Diag.xOverTempMC2			:= 		wEL2904_TempErr.1;
				q_stEL2904_Diag.xOverTempOutputBoard	:= 		wEL2904_TempErr.2;
				q_stEL2904_Diag.xUnderTempMC1			:= 		wEL2904_TempErr.3;
				q_stEL2904_Diag.xUnderTempMC2			:= 		wEL2904_TempErr.4;
				q_stEL2904_Diag.xUnderTempOutputBoard	:= 		wEL2904_TempErr.5;
				q_stEL2904_Diag.xTempDiffOutputBoard	:= 		wEL2904_TempErr.6;
				q_stEL2904_Diag.xTempDiff_MC1MC2		:= 		wEL2904_TempErr.7;
			ELSIF i_xLatchedMessageReset THEN
				q_stEL2904_Diag.xOverTempMC1 			:= FALSE;
				q_stEL2904_Diag.xOverTempMC2 			:= FALSE;
				q_stEL2904_Diag.xOverTempOutputBoard 	:= FALSE;
				q_stEL2904_Diag.xUnderTempMC1 			:= FALSE;
				q_stEL2904_Diag.xUnderTempMC2 			:= FALSE;
				q_stEL2904_Diag.xUnderTempOutputBoard 	:= FALSE;
				q_stEL2904_Diag.xTempDiffOutputBoard 	:= FALSE;
				q_stEL2904_Diag.xTempDiff_MC1MC2 		:= FALSE;
			END_IF
			fbCoERead.bExecute := FALSE;
			q_sErrorDescription := 'No Error';
			iState := iState + 10;
			IF fbCoERead.bError THEN
				q_sErrorDescription := 'EL2904 Output Error Acknowledge Active/Inactive Read Error';
			END_IF
		END_IF	

	300://Set Parameters to read Connection State of the EL2904.	
		fbCoERead.nSubIndex	:= 	1;
		fbCoERead.nIndex	:= 	16#A000;
		fbCoERead.pDstBuf	:= 	ADR(iEL2904_ConnectionState);
		fbCoERead.cbBufLen	:= 	SIZEOF(iEL2904_ConnectionState);
		fbCoERead.bExecute	:= 	TRUE;		
		iState := iState + 10;	
			
	310:// Evaluate read Connection State of the EL2904.			
		IF NOT fbCoERead.bBusy THEN
			IF iEL2904_ConnectionState = 0 THEN
				q_stEL2904_Diag.sConnectionState := 'Reset State';
			ELSIF iEL2904_ConnectionState = 1 THEN
				q_stEL2904_Diag.sConnectionState := 'Session State';
			ELSIF iEL2904_ConnectionState = 2 THEN
				q_stEL2904_Diag.sConnectionState := 'Connection State';
			ELSIF iEL2904_ConnectionState = 3 THEN
				q_stEL2904_Diag.sConnectionState := 'Parameter State';
			ELSIF iEL2904_ConnectionState = 4 THEN
				q_stEL2904_Diag.sConnectionState := 'Data State';
			ELSIF iEL2904_ConnectionState = 5 THEN
				q_stEL2904_Diag.sConnectionState := 'Failsafe State';
			ELSE
				q_stEL2904_Diag.sConnectionState := 'Undefined State';
			END_IF
			fbCoERead.bExecute := FALSE;
			q_sErrorDescription := 'No Error';
			iState := 0;
			IF fbCoERead.bError THEN
				q_sErrorDescription := 'EL2904 Connection State - Read Error';
			END_IF
		END_IF	
END_CASE

// FB_EcCoESdoRead for all CoE reads.
fbCoERead(
	sNetId:= i_sNetId, 
	nSlaveAddr:= i_nSlaveAddr, 
	nSubIndex:= , 
	nIndex:= , 
	pDstBuf:= , 
	cbBufLen:= , 
	bExecute:= , 
	tTimeout:= T#2S, 
	bBusy=> , 
	bError=> q_xError, 
	nErrId=> q_nErrorID);

// If any of above errors exist set stEL2904_Info.xEL2904Error TRUE.
IF NOT q_stEL2904_Diag.xExternalSupplyOrCrossCircuitError1 OR
	q_stEL2904_Diag.xExternalSupplyOrCrossCircuitError2 OR
	q_stEL2904_Diag.xExternalSupplyOrCrossCircuitError3 OR
	q_stEL2904_Diag.xExternalSupplyOrCrossCircuitError4 OR
	q_stEL2904_Diag.xLoadError1 OR
	q_stEL2904_Diag.xLoadError2 OR
	q_stEL2904_Diag.xLoadError3 OR
	q_stEL2904_Diag.xLoadError4 OR
	q_stEL2904_Diag.xOverTempMC1 OR
	q_stEL2904_Diag.xOverTempMC2 OR
	q_stEL2904_Diag.xOverTempOutputBoard OR
	q_stEL2904_Diag.xPowerRailSupplyVoltHighError OR
	q_stEL2904_Diag.xPowerRailSupplyVoltLowError OR
	q_stEL2904_Diag.xTempDiff_MC1MC2 OR
	q_stEL2904_Diag.xTempDiffOutputBoard OR
	q_stEL2904_Diag.xUnderTempMC1 OR
	q_stEL2904_Diag.xUnderTempMC2 OR
	q_stEL2904_Diag.xUnderTempOutputBoard THEN
		q_stEL2904_Diag.xEL2904Error := FALSE;
ELSIF q_stEL2904_Diag.xExternalSupplyOrCrossCircuitError1 OR
	q_stEL2904_Diag.xExternalSupplyOrCrossCircuitError2 OR
	q_stEL2904_Diag.xExternalSupplyOrCrossCircuitError3 OR
	q_stEL2904_Diag.xExternalSupplyOrCrossCircuitError4 OR
	q_stEL2904_Diag.xLoadError1 OR
	q_stEL2904_Diag.xLoadError2 OR
	q_stEL2904_Diag.xLoadError3 OR
	q_stEL2904_Diag.xLoadError4 OR
	q_stEL2904_Diag.xOverTempMC1 OR
	q_stEL2904_Diag.xOverTempMC2 OR
	q_stEL2904_Diag.xOverTempOutputBoard OR
	q_stEL2904_Diag.xPowerRailSupplyVoltHighError OR
	q_stEL2904_Diag.xPowerRailSupplyVoltLowError OR
	q_stEL2904_Diag.xTempDiff_MC1MC2 OR
	q_stEL2904_Diag.xTempDiffOutputBoard OR
	q_stEL2904_Diag.xUnderTempMC1 OR
	q_stEL2904_Diag.xUnderTempMC2 OR
	q_stEL2904_Diag.xUnderTempOutputBoard THEN
		q_stEL2904_Diag.xEL2904Error := TRUE;
END_IF

END_FUNCTION_BLOCK

// POUs/HardwareFBs/FB_EK1914Diagnostics
(*=====================================================================
Beckhoff Automation LLC
Copyright 2015 All Rights Reserved
=======================================================================
Description: 
This Program has been supplied by Beckhoff Automation As-Is and is intended only as an example implementation. 
Functionality is not guaranteed. 
This Function Block reads all status and error information known at time of creation of the EK1914.
---------------------------------------------------------------------------------------------------------------
History:
Date		Version			Author							Comment
---------------------------------------------------------------------------------------------------------------
07.08.15	0.10		Jason Erickson				Initial Library Creation.
07.20.15	0.11		Jason Ericskon				Added CoE Read for TwinSAFE Connection State.
08.28.15	0.20		Jason Erickson				Code optimization to eliminate timed data reads.
09.18.15	0.2.1		Jason Erickson				Added new error codes 0x6000 - 0x6002 and Connection Status to the AX5805.
09.24.15	0.2.2		Jason Erickson				Corrected inability to update CASE in FB_EL1904Diagnostics and FB_EL2904Diagnostics.
10.30.15	0.2.3		Jason Erickson				Modified Diagnostic Structure names for ease of use.
*)
FUNCTION_BLOCK FB_EK1914Diagnostics
VAR_INPUT
	i_sNetId: STRING;				// EtherCAT Master Device Net ID.
	i_nSlaveAddr: UINT;				// Slave Address of the EK1914.
	i_xLatchedMessageReset: BOOL;	// Reset the internal Latched Data FBs.
END_VAR
VAR_OUTPUT
	q_stEK1914_Diag: ST_EK1914_DIAGNOSTICS;	// Output structure containing all Status and Diagnostic information.
	q_xError: BOOL;							// Internal Function Block error. 
	q_udiErrorID: UDINT;					// Internal Function Block error number when the q_xError is set. 
	q_sErrorDescription: STRING;			// Internal Function Block error description when the q_xError is set.
END_VAR
VAR
// Case Statement
	iState: INT;
// FB_EcCoESdoRead for all CoE reads.
	fbCoERead: FB_EcCoESdoRead;
// Variable to hold data for evaluation, Micro Controller (MC1) 3.3v Nominal Voltage (mV) INPUT of the EK1914.
	wEK1914_MC1_3300mV: WORD;
// Variable to hold data for evaluation, Micro Controller (MC2) 3.3v Nominal Voltage (mV) INPUT of the EK1914.
	wEK1914_MC2_3300mV: WORD;
// Variable to hold data for evaluation, Standard Output Active/Inactive of the EK1914.
		(* Standard outputs can be used to directly Enable/Disable a TwinSAFE output
	   		if this feature is ACTIVE (Not to Turn it ON/OFF, Allow it or not to turn ON!!! *)
	bEK1914_StandardOuts: BYTE;
// Variable to hold data for evaluation, Test Pulses Active/Inactive of the EK1914.
		(* Used to determine TwinSAFE output wiring is correct *)
	bEK1914_TestP: BYTE;
// Variable to hold data for evaluation, Output Error Acknowledge Active/Inactive of the EK1914.
		(* Used to reset TwinSAFE output errors instead of forcing a cycle power
			for a TwinSAFE output error. *)
	bEK1914_ErrAck: BYTE;
// Variable to hold data for evaluation, Sensor Tests Active/Inactive Channel 1 of the EK1914.
	iEK1914_STActive1: BOOL;
// Variable to hold data for evaluation, Sensor Tests Active/Inactive Channel 2 of the EK1914.
	iEK1914_STActive2: BOOL;
// Variable to hold data for evaluation, Logic setting of Channels 1 and 2 of the EK1914.
	bEK1914_Logic1_2: BYTE;
// Variable to hold data for evaluation, Sensor Tests Errors of the EK1914.
	wEK1914_SenT: WORD;
// Variable to hold data for evaluation, Two-Channel Evaluation Error - Diagnostic object 800E:0B
		(* The two channels contradict each other (not same value). *)
	wEK1914_2CHEval: WORD;
// Variable to hold data for evaluation, Error In Safety Mat Operating Mode: Input Pair Disagree - Diagnostic object 800E:0C
		(* Input pairs not in the same state (not same value). *)
	wEK1914_SMiPair: WORD;
// Variable to hold data for evaluation, Error In Safety Mat Operating Mode: External Supply (No test pulses) - Diagnostic object 800E:0D
		(* External supply detected (Input channel not getting test pulses). *)
	wEK1914_SMExtSupply: WORD;
// Variable to hold data for evaluation, Error At The Output MC1 of the EK1914.
		(* External supply or cross-circuit Error Open Load, Current Below 20mA, OR Current Above Maximum Value OF 500mA. *)
	wEK1914_OutErrMC1: WORD;
// Variable to hold data for evaluation, Error At The Output MC2 of the EK1914.
		(* External supply or cross-circuit Error Open Load, Current Below 20mA, OR Current Above Maximum Value OF 500mA. *)
	wEK1914_OutErrMC2: WORD;
// Variable to hold data for evaluation, Connection State of the EK1914.
	iEK1914_ConnectionState: INT;
END_VAR

CASE iState OF
	0:// Set Parameters to read the Serial Number of the EK1914.		
		fbCoERead.nSubIndex := 16#02;
		fbCoERead.nIndex 	:= 16#F980;
		fbCoERead.pDstBuf	:= 	ADR(q_stEK1914_Diag.dwSerialNumber);
		fbCoERead.cbBufLen	:= 	SIZEOF(q_stEK1914_Diag.dwSerialNumber);
		fbCoERead.bExecute	:= TRUE;
		iState := iState + 10;
		
	10:// Evaluate read of the Serial Number of the EL1914.
		IF NOT fbCoERead.bBusy THEN
			fbCoERead.bExecute	:= FALSE;
			q_sErrorDescription := 'No Error';
			iState := iState + 10;
		ELSIF fbCoERead.bError THEN
			q_sErrorDescription := 'EK1914 Serial Number - Read Error';
		END_IF
	
	20:// Set Parameters to read the DIP Switch Setting of the EK1914.		
		fbCoERead.nSubIndex := 16#01;
		fbCoERead.nIndex 	:= 16#F980;
		fbCoERead.pDstBuf	:= 	ADR(q_stEK1914_Diag.wDipSwitch);
		fbCoERead.cbBufLen	:= 	SIZEOF(q_stEK1914_Diag.wDipSwitch);
		fbCoERead.bExecute	:= TRUE;
		iState := iState + 10;
			
	30:// Evaluate read of the DIP Switch setting of the EK1914.	
		IF NOT fbCoERead.bBusy THEN
			fbCoERead.bExecute	:= FALSE;
			q_sErrorDescription := 'No Error';
			iState := iState + 10;
		ELSIF fbCoERead.bError THEN
			q_sErrorDescription := 'EK1914 DIP Switch - Read Error';
		END_IF
	
	40:// Set Parameters to read the Hardware Version of the EK1914.	
		fbCoERead.nSubIndex := 0;
		fbCoERead.nIndex 	:= 16#1009;
		fbCoERead.pDstBuf	:= 	ADR(q_stEK1914_Diag.sHwVersion);
		fbCoERead.cbBufLen	:= 	SIZEOF(q_stEK1914_Diag.sHwVersion);
		fbCoERead.bExecute	:= TRUE;
		iState := iState + 10;
		
	50:// Evaluate read of the Hardware Version of the EK1914.
		IF NOT fbCoERead.bBusy THEN
			fbCoERead.bExecute	:= FALSE;
			q_sErrorDescription := 'No Error';
			iState := iState + 10;
		ELSIF fbCoERead.bError THEN
			q_sErrorDescription := 'EK1914 Hardware Version - Read Error';
		END_IF	

	60:// Set Parameters to read the Software Version (firmware) of the EK1914.
		fbCoERead.nSubIndex := 0;
		fbCoERead.nIndex 	:= 16#100A;
		fbCoERead.pDstBuf	:= 	ADR(q_stEK1914_Diag.sFwVersion);
		fbCoERead.cbBufLen	:= 	SIZEOF(q_stEK1914_Diag.sFwVersion);
		fbCoERead.bExecute	:= TRUE;
		iState := iState + 10;

	70:// Evaluate read of the Software Version (firmware) of the EK1914.
		IF NOT fbCoERead.bBusy THEN
			fbCoERead.bExecute	:= FALSE;
			q_sErrorDescription := 'No Error';
			iState := iState + 10;
		ELSIF fbCoERead.bError THEN
			q_sErrorDescription := 'EK1914 Software Version (firmware) - Read Error';
		END_IF	
		
	80:// Set Parameters to read the Micro Controller (MC1) Temperature in DegC of the EK1914.		
		fbCoERead.nSubIndex := 16#01;
		fbCoERead.nIndex 	:= 16#FA80;
		fbCoERead.pDstBuf	:= 	ADR(q_stEK1914_Diag.wMC1Temp);
		fbCoERead.cbBufLen	:= 	SIZEOF(q_stEK1914_Diag.wMC1Temp);
		fbCoERead.bExecute	:= TRUE;
		iState := iState + 10;
	
	90:// Evaluate read of the Micro Controller (MC1) Temperature in DegC of the EK1914.	
		IF NOT fbCoERead.bBusy THEN
			fbCoERead.bExecute	:= FALSE;
			q_sErrorDescription := 'No Error';
			iState := iState + 10;
		ELSIF fbCoERead.bError THEN
			q_sErrorDescription := 'EK1914 MC1 Temp - Read Error';
		END_IF	

	100:// Set Parameters to read the Micro Controller (MC2) Temperature in DegC of the EK1914.
		fbCoERead.nSubIndex := 16#02;
		fbCoERead.nIndex 	:= 16#FA80;
		fbCoERead.pDstBuf	:= 	ADR(q_stEK1914_Diag.wMC2Temp);
		fbCoERead.cbBufLen	:= 	SIZEOF(q_stEK1914_Diag.wMC2Temp);
		fbCoERead.bExecute	:= TRUE;
		iState := iState + 10;
	
	110:// Evaluate read of the Micro Controller (MC2) Temperature in DegC of the EK1914.
		IF NOT fbCoERead.bBusy THEN
			fbCoERead.bExecute	:= FALSE;
			q_sErrorDescription := 'No Error';
			iState := iState + 10;
		ELSIF fbCoERead.bError THEN
			q_sErrorDescription := 'EK1914 MC2 Temp - Read Error';
		END_IF	

